//     PlcTask Inputs/GVL_iXlinker.EtherCAT_Master_BKCUCX.TcTerminals210_EK1100_1.TcTerminals210_1BK1250.A_0265_KM_2774_4_Ch_Blinds_control_CM_Inputs_230V_AC_1A.Channel_1.State <-> Channel 1/State
//     PlcTask Inputs/GVL_iXlinker.EtherCAT_Master_BKCUCX.TcTerminals210_EK1100_1.TcTerminals210_1BK1250.A_0265_KM_2774_4_Ch_Blinds_control_CM_Inputs_230V_AC_1A.Channel_1.Data_In <-> Channel 1/Data In
//     PlcTask Outputs/GVL_iXlinker.EtherCAT_Master_BKCUCX.TcTerminals210_EK1100_1.TcTerminals210_1BK1250.A_0265_KM_2774_4_Ch_Blinds_control_CM_Inputs_230V_AC_1A.Channel_1.Ctrl <-> Channel 1/Ctrl
//     PlcTask Outputs/GVL_iXlinker.EtherCAT_Master_BKCUCX.TcTerminals210_EK1100_1.TcTerminals210_1BK1250.A_0265_KM_2774_4_Ch_Blinds_control_CM_Inputs_230V_AC_1A.Channel_1.Data_Out <-> Channel 1/Data Out
//   PLC/PLC Instance <-> EtherCAT Master BKCUCX/TcTerminals210_EK1100_1/TcTerminals210_1BK1250/A_0266(Buerkert valve island 2 channels)
//     PlcTask Outputs/GVL_iXlinker.EtherCAT_Master_BKCUCX.TcTerminals210_EK1100_1.TcTerminals210_1BK1250.A_0266_Buerkert_valve_island_2_channels.Channel_1.Output <-> Channel 1/Output
//     PlcTask Outputs/GVL_iXlinker.EtherCAT_Master_BKCUCX.TcTerminals210_EK1100_1.TcTerminals210_1BK1250.A_0266_Buerkert_valve_island_2_channels.Channel_2.Output <-> Channel 2/Output
//   PLC/PLC Instance <-> EtherCAT Master BKCUCX/TcTerminals210_EK1100_1/TcTerminals210_1BK1250/A_0267(Buerkert valve island 4 channels)
//     PlcTask Outputs/GVL_iXlinker.EtherCAT_Master_BKCUCX.TcTerminals210_EK1100_1.TcTerminals210_1BK1250.A_0267_Buerkert_valve_island_4_channels.Channel_1.Output <-> Channel 1/Output
//     PlcTask Outputs/GVL_iXlinker.EtherCAT_Master_BKCUCX.TcTerminals210_EK1100_1.TcTerminals210_1BK1250.A_0267_Buerkert_valve_island_4_channels.Channel_2.Output <-> Channel 2/Output
//     PlcTask Outputs/GVL_iXlinker.EtherCAT_Master_BKCUCX.TcTerminals210_EK1100_1.TcTerminals210_1BK1250.A_0267_Buerkert_valve_island_4_channels.Channel_3.Output <-> Channel 3/Output
//     PlcTask Outputs/GVL_iXlinker.EtherCAT_Master_BKCUCX.TcTerminals210_EK1100_1.TcTerminals210_1BK1250.A_0267_Buerkert_valve_island_4_channels.Channel_4.Output <-> Channel 4/Output
//   PLC/PLC Instance <-> EtherCAT Master BKCUCX/TcTerminals210_EK1100_1/TcTerminals210_1BK1250/A_0268(Buerkert valve island 8 channels)
//     PlcTask Outputs/GVL_iXlinker.EtherCAT_Master_BKCUCX.TcTerminals210_EK1100_1.TcTerminals210_1BK1250.A_0268_Buerkert_valve_island_8_channels.Channel_1.Output <-> Channel 1/Output
//     PlcTask Outputs/GVL_iXlinker.EtherCAT_Master_BKCUCX.TcTerminals210_EK1100_1.TcTerminals210_1BK1250.A_0268_Buerkert_valve_island_8_channels.Channel_2.Output <-> Channel 2/Output
//     PlcTask Outputs/GVL_iXlinker.EtherCAT_Master_BKCUCX.TcTerminals210_EK1100_1.TcTerminals210_1BK1250.A_0268_Buerkert_valve_island_8_channels.Channel_3.Output <-> Channel 3/Output
//     PlcTask Outputs/GVL_iXlinker.EtherCAT_Master_BKCUCX.TcTerminals210_EK1100_1.TcTerminals210_1BK1250.A_0268_Buerkert_valve_island_8_channels.Channel_4.Output <-> Channel 4/Output
//     PlcTask Outputs/GVL_iXlinker.EtherCAT_Master_BKCUCX.TcTerminals210_EK1100_1.TcTerminals210_1BK1250.A_0268_Buerkert_valve_island_8_channels.Channel_5.Output <-> Channel 5/Output
//     PlcTask Outputs/GVL_iXlinker.EtherCAT_Master_BKCUCX.TcTerminals210_EK1100_1.TcTerminals210_1BK1250.A_0268_Buerkert_valve_island_8_channels.Channel_6.Output <-> Channel 6/Output
//     PlcTask Outputs/GVL_iXlinker.EtherCAT_Master_BKCUCX.TcTerminals210_EK1100_1.TcTerminals210_1BK1250.A_0268_Buerkert_valve_island_8_channels.Channel_7.Output <-> Channel 7/Output
//     PlcTask Outputs/GVL_iXlinker.EtherCAT_Master_BKCUCX.TcTerminals210_EK1100_1.TcTerminals210_1BK1250.A_0268_Buerkert_valve_island_8_channels.Channel_8.Output <-> Channel 8/Output
//   PLC/PLC Instance <-> EtherCAT Master BKCUCX/TcTerminals210_EK1100_1/TcTerminals210_1BK1250/A_0269(KL 3001, 1 Ch. ana. Input (-10V/0...10V))
//     PlcTask Inputs/GVL_iXlinker.EtherCAT_Master_BKCUCX.TcTerminals210_EK1100_1.TcTerminals210_1BK1250.A_0269_KL_3001_1_Ch_ana_Input_10V_0_10V.Channel_1.State <-> Channel 1/State
//     PlcTask Inputs/GVL_iXlinker.EtherCAT_Master_BKCUCX.TcTerminals210_EK1100_1.TcTerminals210_1BK1250.A_0269_KL_3001_1_Ch_ana_Input_10V_0_10V.Channel_1.Data_In <-> Channel 1/Data In
//     PlcTask Outputs/GVL_iXlinker.EtherCAT_Master_BKCUCX.TcTerminals210_EK1100_1.TcTerminals210_1BK1250.A_0269_KL_3001_1_Ch_ana_Input_10V_0_10V.Channel_1.Ctrl <-> Channel 1/Ctrl
//     PlcTask Outputs/GVL_iXlinker.EtherCAT_Master_BKCUCX.TcTerminals210_EK1100_1.TcTerminals210_1BK1250.A_0269_KL_3001_1_Ch_ana_Input_10V_0_10V.Channel_1.Data_Out <-> Channel 1/Data Out
//   PLC/PLC Instance <-> EtherCAT Master BKCUCX/TcTerminals210_EK1100_1/TcTerminals210_1BK1250/A_0271(KL 3002, 2 Ch. ana. Input (-10V/0...10V))
//     PlcTask Inputs/GVL_iXlinker.EtherCAT_Master_BKCUCX.TcTerminals210_EK1100_1.TcTerminals210_1BK1250.A_0271_KL_3002_2_Ch_ana_Input_10V_0_10V.Channel_1.State <-> Channel 1/State
//     PlcTask Inputs/GVL_iXlinker.EtherCAT_Master_BKCUCX.TcTerminals210_EK1100_1.TcTerminals210_1BK1250.A_0271_KL_3002_2_Ch_ana_Input_10V_0_10V.Channel_2.State <-> Channel 2/State
//     PlcTask Inputs/GVL_iXlinker.EtherCAT_Master_BKCUCX.TcTerminals210_EK1100_1.TcTerminals210_1BK1250.A_0271_KL_3002_2_Ch_ana_Input_10V_0_10V.Channel_1.Data_In <-> Channel 1/Data In
//     PlcTask Inputs/GVL_iXlinker.EtherCAT_Master_BKCUCX.TcTerminals210_EK1100_1.TcTerminals210_1BK1250.A_0271_KL_3002_2_Ch_ana_Input_10V_0_10V.Channel_2.Data_In <-> Channel 2/Data In
//     PlcTask Outputs/GVL_iXlinker.EtherCAT_Master_BKCUCX.TcTerminals210_EK1100_1.TcTerminals210_1BK1250.A_0271_KL_3002_2_Ch_ana_Input_10V_0_10V.Channel_1.Ctrl <-> Channel 1/Ctrl
//     PlcTask Outputs/GVL_iXlinker.EtherCAT_Master_BKCUCX.TcTerminals210_EK1100_1.TcTerminals210_1BK1250.A_0271_KL_3002_2_Ch_ana_Input_10V_0_10V.Channel_2.Ctrl <-> Channel 2/Ctrl
//     PlcTask Outputs/GVL_iXlinker.EtherCAT_Master_BKCUCX.TcTerminals210_EK1100_1.TcTerminals210_1BK1250.A_0271_KL_3002_2_Ch_ana_Input_10V_0_10V.Channel_1.Data_Out <-> Channel 1/Data Out
//     PlcTask Outputs/GVL_iXlinker.EtherCAT_Master_BKCUCX.TcTerminals210_EK1100_1.TcTerminals210_1BK1250.A_0271_KL_3002_2_Ch_ana_Input_10V_0_10V.Channel_2.Data_Out <-> Channel 2/Data Out
//   PLC/PLC Instance <-> EtherCAT Master BKCUCX/TcTerminals210_EK1100_1/TcTerminals210_1BK1250/A_0273(KL 3011, 1 Ch. ana. Input (0 - 20mA))
//     PlcTask Inputs/GVL_iXlinker.EtherCAT_Master_BKCUCX.TcTerminals210_EK1100_1.TcTerminals210_1BK1250.A_0273_KL_3011_1_Ch_ana_Input_0_20mA.Channel_1.State <-> Channel 1/State
//     PlcTask Inputs/GVL_iXlinker.EtherCAT_Master_BKCUCX.TcTerminals210_EK1100_1.TcTerminals210_1BK1250.A_0273_KL_3011_1_Ch_ana_Input_0_20mA.Channel_1.Data_In <-> Channel 1/Data In
//     PlcTask Outputs/GVL_iXlinker.EtherCAT_Master_BKCUCX.TcTerminals210_EK1100_1.TcTerminals210_1BK1250.A_0273_KL_3011_1_Ch_ana_Input_0_20mA.Channel_1.Ctrl <-> Channel 1/Ctrl
//     PlcTask Outputs/GVL_iXlinker.EtherCAT_Master_BKCUCX.TcTerminals210_EK1100_1.TcTerminals210_1BK1250.A_0273_KL_3011_1_Ch_ana_Input_0_20mA.Channel_1.Data_Out <-> Channel 1/Data Out
//   PLC/PLC Instance <-> EtherCAT Master BKCUCX/TcTerminals210_EK1100_1/TcTerminals210_1BK1250/A_0275(KL 3012, 2 Ch. ana. Input (0 - 20mA))
//     PlcTask Inputs/GVL_iXlinker.EtherCAT_Master_BKCUCX.TcTerminals210_EK1100_1.TcTerminals210_1BK1250.A_0275_KL_3012_2_Ch_ana_Input_0_20mA.Channel_1.State <-> Channel 1/State
//     PlcTask Inputs/GVL_iXlinker.EtherCAT_Master_BKCUCX.TcTerminals210_EK1100_1.TcTerminals210_1BK1250.A_0275_KL_3012_2_Ch_ana_Input_0_20mA.Channel_2.State <-> Channel 2/State
//     PlcTask Inputs/GVL_iXlinker.EtherCAT_Master_BKCUCX.TcTerminals210_EK1100_1.TcTerminals210_1BK1250.A_0275_KL_3012_2_Ch_ana_Input_0_20mA.Channel_1.Data_In <-> Channel 1/Data In
//     PlcTask Inputs/GVL_iXlinker.EtherCAT_Master_BKCUCX.TcTerminals210_EK1100_1.TcTerminals210_1BK1250.A_0275_KL_3012_2_Ch_ana_Input_0_20mA.Channel_2.Data_In <-> Channel 2/Data In
//     PlcTask Outputs/GVL_iXlinker.EtherCAT_Master_BKCUCX.TcTerminals210_EK1100_1.TcTerminals210_1BK1250.A_0275_KL_3012_2_Ch_ana_Input_0_20mA.Channel_1.Ctrl <-> Channel 1/Ctrl
//     PlcTask Outputs/GVL_iXlinker.EtherCAT_Master_BKCUCX.TcTerminals210_EK1100_1.TcTerminals210_1BK1250.A_0275_KL_3012_2_Ch_ana_Input_0_20mA.Channel_2.Ctrl <-> Channel 2/Ctrl
//     PlcTask Outputs/GVL_iXlinker.EtherCAT_Master_BKCUCX.TcTerminals210_EK1100_1.TcTerminals210_1BK1250.A_0275_KL_3012_2_Ch_ana_Input_0_20mA.Channel_1.Data_Out <-> Channel 1/Data Out
//     PlcTask Outputs/GVL_iXlinker.EtherCAT_Master_BKCUCX.TcTerminals210_EK1100_1.TcTerminals210_1BK1250.A_0275_KL_3012_2_Ch_ana_Input_0_20mA.Channel_2.Data_Out <-> Channel 2/Data Out
//   PLC/PLC Instance <-> EtherCAT Master BKCUCX/TcTerminals210_EK1100_1/TcTerminals210_1BK1250/A_0277(KL 3021, 1 Ch. ana. Input (4 - 20mA))
//     PlcTask Inputs/GVL_iXlinker.EtherCAT_Master_BKCUCX.TcTerminals210_EK1100_1.TcTerminals210_1BK1250.A_0277_KL_3021_1_Ch_ana_Input_4_20mA.Channel_1.State <-> Channel 1/State
//     PlcTask Inputs/GVL_iXlinker.EtherCAT_Master_BKCUCX.TcTerminals210_EK1100_1.TcTerminals210_1BK1250.A_0277_KL_3021_1_Ch_ana_Input_4_20mA.Channel_1.Data_In <-> Channel 1/Data In
//     PlcTask Outputs/GVL_iXlinker.EtherCAT_Master_BKCUCX.TcTerminals210_EK1100_1.TcTerminals210_1BK1250.A_0277_KL_3021_1_Ch_ana_Input_4_20mA.Channel_1.Ctrl <-> Channel 1/Ctrl
//     PlcTask Outputs/GVL_iXlinker.EtherCAT_Master_BKCUCX.TcTerminals210_EK1100_1.TcTerminals210_1BK1250.A_0277_KL_3021_1_Ch_ana_Input_4_20mA.Channel_1.Data_Out <-> Channel 1/Data Out
//   PLC/PLC Instance <-> EtherCAT Master BKCUCX/TcTerminals210_EK1100_1/TcTerminals210_1BK1250/A_0279(KL 3022, 2 Ch. ana. Input (4 - 20mA))
//     PlcTask Inputs/GVL_iXlinker.EtherCAT_Master_BKCUCX.TcTerminals210_EK1100_1.TcTerminals210_1BK1250.A_0279_KL_3022_2_Ch_ana_Input_4_20mA.Channel_1.State <-> Channel 1/State
//     PlcTask Inputs/GVL_iXlinker.EtherCAT_Master_BKCUCX.TcTerminals210_EK1100_1.TcTerminals210_1BK1250.A_0279_KL_3022_2_Ch_ana_Input_4_20mA.Channel_2.State <-> Channel 2/State
//     PlcTask Inputs/GVL_iXlinker.EtherCAT_Master_BKCUCX.TcTerminals210_EK1100_1.TcTerminals210_1BK1250.A_0279_KL_3022_2_Ch_ana_Input_4_20mA.Channel_1.Data_In <-> Channel 1/Data In
//     PlcTask Inputs/GVL_iXlinker.EtherCAT_Master_BKCUCX.TcTerminals210_EK1100_1.TcTerminals210_1BK1250.A_0279_KL_3022_2_Ch_ana_Input_4_20mA.Channel_2.Data_In <-> Channel 2/Data In
//     PlcTask Outputs/GVL_iXlinker.EtherCAT_Master_BKCUCX.TcTerminals210_EK1100_1.TcTerminals210_1BK1250.A_0279_KL_3022_2_Ch_ana_Input_4_20mA.Channel_1.Ctrl <-> Channel 1/Ctrl
//     PlcTask Outputs/GVL_iXlinker.EtherCAT_Master_BKCUCX.TcTerminals210_EK1100_1.TcTerminals210_1BK1250.A_0279_KL_3022_2_Ch_ana_Input_4_20mA.Channel_2.Ctrl <-> Channel 2/Ctrl
//     PlcTask Outputs/GVL_iXlinker.EtherCAT_Master_BKCUCX.TcTerminals210_EK1100_1.TcTerminals210_1BK1250.A_0279_KL_3022_2_Ch_ana_Input_4_20mA.Channel_1.Data_Out <-> Channel 1/Data Out
//     PlcTask Outputs/GVL_iXlinker.EtherCAT_Master_BKCUCX.TcTerminals210_EK1100_1.TcTerminals210_1BK1250.A_0279_KL_3022_2_Ch_ana_Input_4_20mA.Channel_2.Data_Out <-> Channel 2/Data Out
//   PLC/PLC Instance <-> EtherCAT Master BKCUCX/TcTerminals210_EK1100_1/TcTerminals210_1BK1250/A_0281(KL 3041, 1 Ch. ana. Input with Power (0 - 20mA))
//     PlcTask Inputs/GVL_iXlinker.EtherCAT_Master_BKCUCX.TcTerminals210_EK1100_1.TcTerminals210_1BK1250.A_0281_KL_3041_1_Ch_ana_Input_with_Power_0_20mA.Channel_1.State <-> Channel 1/State
//     PlcTask Inputs/GVL_iXlinker.EtherCAT_Master_BKCUCX.TcTerminals210_EK1100_1.TcTerminals210_1BK1250.A_0281_KL_3041_1_Ch_ana_Input_with_Power_0_20mA.Channel_1.Data_In <-> Channel 1/Data In
//     PlcTask Outputs/GVL_iXlinker.EtherCAT_Master_BKCUCX.TcTerminals210_EK1100_1.TcTerminals210_1BK1250.A_0281_KL_3041_1_Ch_ana_Input_with_Power_0_20mA.Channel_1.Ctrl <-> Channel 1/Ctrl
//     PlcTask Outputs/GVL_iXlinker.EtherCAT_Master_BKCUCX.TcTerminals210_EK1100_1.TcTerminals210_1BK1250.A_0281_KL_3041_1_Ch_ana_Input_with_Power_0_20mA.Channel_1.Data_Out <-> Channel 1/Data Out
//   PLC/PLC Instance <-> EtherCAT Master BKCUCX/TcTerminals210_EK1100_1/TcTerminals210_1BK1250/A_0283(KL 3042, 2 Ch. ana. Input with Power (0 - 20mA))
//     PlcTask Inputs/GVL_iXlinker.EtherCAT_Master_BKCUCX.TcTerminals210_EK1100_1.TcTerminals210_1BK1250.A_0283_KL_3042_2_Ch_ana_Input_with_Power_0_20mA.Channel_1.State <-> Channel 1/State
//     PlcTask Inputs/GVL_iXlinker.EtherCAT_Master_BKCUCX.TcTerminals210_EK1100_1.TcTerminals210_1BK1250.A_0283_KL_3042_2_Ch_ana_Input_with_Power_0_20mA.Channel_2.State <-> Channel 2/State
//     PlcTask Inputs/GVL_iXlinker.EtherCAT_Master_BKCUCX.TcTerminals210_EK1100_1.TcTerminals210_1BK1250.A_0283_KL_3042_2_Ch_ana_Input_with_Power_0_20mA.Channel_1.Data_In <-> Channel 1/Data In
//     PlcTask Inputs/GVL_iXlinker.EtherCAT_Master_BKCUCX.TcTerminals210_EK1100_1.TcTerminals210_1BK1250.A_0283_KL_3042_2_Ch_ana_Input_with_Power_0_20mA.Channel_2.Data_In <-> Channel 2/Data In
//     PlcTask Outputs/GVL_iXlinker.EtherCAT_Master_BKCUCX.TcTerminals210_EK1100_1.TcTerminals210_1BK1250.A_0283_KL_3042_2_Ch_ana_Input_with_Power_0_20mA.Channel_1.Ctrl <-> Channel 1/Ctrl
//     PlcTask Outputs/GVL_iXlinker.EtherCAT_Master_BKCUCX.TcTerminals210_EK1100_1.TcTerminals210_1BK1250.A_0283_KL_3042_2_Ch_ana_Input_with_Power_0_20mA.Channel_2.Ctrl <-> Channel 2/Ctrl
//     PlcTask Outputs/GVL_iXlinker.EtherCAT_Master_BKCUCX.TcTerminals210_EK1100_1.TcTerminals210_1BK1250.A_0283_KL_3042_2_Ch_ana_Input_with_Power_0_20mA.Channel_1.Data_Out <-> Channel 1/Data Out
//     PlcTask Outputs/GVL_iXlinker.EtherCAT_Master_BKCUCX.TcTerminals210_EK1100_1.TcTerminals210_1BK1250.A_0283_KL_3042_2_Ch_ana_Input_with_Power_0_20mA.Channel_2.Data_Out <-> Channel 2/Data Out
//   PLC/PLC Instance <-> EtherCAT Master BKCUCX/TcTerminals210_EK1100_1/TcTerminals210_1BK1250/A_0285(KL 3044, 4 Ch. ana. Input with Power (0 - 20mA))
//     PlcTask Inputs/GVL_iXlinker.EtherCAT_Master_BKCUCX.TcTerminals210_EK1100_1.TcTerminals210_1BK1250.A_0285_KL_3044_4_Ch_ana_Input_with_Power_0_20mA.Channel_1.State <-> Channel 1/State
//     PlcTask Inputs/GVL_iXlinker.EtherCAT_Master_BKCUCX.TcTerminals210_EK1100_1.TcTerminals210_1BK1250.A_0285_KL_3044_4_Ch_ana_Input_with_Power_0_20mA.Channel_2.State <-> Channel 2/State
//     PlcTask Inputs/GVL_iXlinker.EtherCAT_Master_BKCUCX.TcTerminals210_EK1100_1.TcTerminals210_1BK1250.A_0285_KL_3044_4_Ch_ana_Input_with_Power_0_20mA.Channel_3.State <-> Channel 3/State
//     PlcTask Inputs/GVL_iXlinker.EtherCAT_Master_BKCUCX.TcTerminals210_EK1100_1.TcTerminals210_1BK1250.A_0285_KL_3044_4_Ch_ana_Input_with_Power_0_20mA.Channel_4.State <-> Channel 4/State
//     PlcTask Inputs/GVL_iXlinker.EtherCAT_Master_BKCUCX.TcTerminals210_EK1100_1.TcTerminals210_1BK1250.A_0285_KL_3044_4_Ch_ana_Input_with_Power_0_20mA.Channel_1.Data_In <-> Channel 1/Data In
//     PlcTask Inputs/GVL_iXlinker.EtherCAT_Master_BKCUCX.TcTerminals210_EK1100_1.TcTerminals210_1BK1250.A_0285_KL_3044_4_Ch_ana_Input_with_Power_0_20mA.Channel_2.Data_In <-> Channel 2/Data In
//     PlcTask Inputs/GVL_iXlinker.EtherCAT_Master_BKCUCX.TcTerminals210_EK1100_1.TcTerminals210_1BK1250.A_0285_KL_3044_4_Ch_ana_Input_with_Power_0_20mA.Channel_3.Data_In <-> Channel 3/Data In
//     PlcTask Inputs/GVL_iXlinker.EtherCAT_Master_BKCUCX.TcTerminals210_EK1100_1.TcTerminals210_1BK1250.A_0285_KL_3044_4_Ch_ana_Input_with_Power_0_20mA.Channel_4.Data_In <-> Channel 4/Data In
//     PlcTask Outputs/GVL_iXlinker.EtherCAT_Master_BKCUCX.TcTerminals210_EK1100_1.TcTerminals210_1BK1250.A_0285_KL_3044_4_Ch_ana_Input_with_Power_0_20mA.Channel_1.Ctrl <-> Channel 1/Ctrl
//     PlcTask Outputs/GVL_iXlinker.EtherCAT_Master_BKCUCX.TcTerminals210_EK1100_1.TcTerminals210_1BK1250.A_0285_KL_3044_4_Ch_ana_Input_with_Power_0_20mA.Channel_2.Ctrl <-> Channel 2/Ctrl
//     PlcTask Outputs/GVL_iXlinker.EtherCAT_Master_BKCUCX.TcTerminals210_EK1100_1.TcTerminals210_1BK1250.A_0285_KL_3044_4_Ch_ana_Input_with_Power_0_20mA.Channel_3.Ctrl <-> Channel 3/Ctrl
//     PlcTask Outputs/GVL_iXlinker.EtherCAT_Master_BKCUCX.TcTerminals210_EK1100_1.TcTerminals210_1BK1250.A_0285_KL_3044_4_Ch_ana_Input_with_Power_0_20mA.Channel_4.Ctrl <-> Channel 4/Ctrl
//     PlcTask Outputs/GVL_iXlinker.EtherCAT_Master_BKCUCX.TcTerminals210_EK1100_1.TcTerminals210_1BK1250.A_0285_KL_3044_4_Ch_ana_Input_with_Power_0_20mA.Channel_1.Data_Out <-> Channel 1/Data Out
//     PlcTask Outputs/GVL_iXlinker.EtherCAT_Master_BKCUCX.TcTerminals210_EK1100_1.TcTerminals210_1BK1250.A_0285_KL_3044_4_Ch_ana_Input_with_Power_0_20mA.Channel_2.Data_Out <-> Channel 2/Data Out
//     PlcTask Outputs/GVL_iXlinker.EtherCAT_Master_BKCUCX.TcTerminals210_EK1100_1.TcTerminals210_1BK1250.A_0285_KL_3044_4_Ch_ana_Input_with_Power_0_20mA.Channel_3.Data_Out <-> Channel 3/Data Out
//     PlcTask Outputs/GVL_iXlinker.EtherCAT_Master_BKCUCX.TcTerminals210_EK1100_1.TcTerminals210_1BK1250.A_0285_KL_3044_4_Ch_ana_Input_with_Power_0_20mA.Channel_4.Data_Out <-> Channel 4/Data Out
//   PLC/PLC Instance <-> EtherCAT Master BKCUCX/TcTerminals210_EK1100_1/TcTerminals210_1BK1250/A_0287(KL 3051, 1 Ch. ana. Input with Power (4 - 20mA))
//     PlcTask Inputs/GVL_iXlinker.EtherCAT_Master_BKCUCX.TcTerminals210_EK1100_1.TcTerminals210_1BK1250.A_0287_KL_3051_1_Ch_ana_Input_with_Power_4_20mA.Channel_1.State <-> Channel 1/State
//     PlcTask Inputs/GVL_iXlinker.EtherCAT_Master_BKCUCX.TcTerminals210_EK1100_1.TcTerminals210_1BK1250.A_0287_KL_3051_1_Ch_ana_Input_with_Power_4_20mA.Channel_1.Data_In <-> Channel 1/Data In
//     PlcTask Outputs/GVL_iXlinker.EtherCAT_Master_BKCUCX.TcTerminals210_EK1100_1.TcTerminals210_1BK1250.A_0287_KL_3051_1_Ch_ana_Input_with_Power_4_20mA.Channel_1.Ctrl <-> Channel 1/Ctrl
//     PlcTask Outputs/GVL_iXlinker.EtherCAT_Master_BKCUCX.TcTerminals210_EK1100_1.TcTerminals210_1BK1250.A_0287_KL_3051_1_Ch_ana_Input_with_Power_4_20mA.Channel_1.Data_Out <-> Channel 1/Data Out
//   PLC/PLC Instance <-> EtherCAT Master BKCUCX/TcTerminals210_EK1100_1/TcTerminals210_1BK1250/A_0289(KL 3052, 2 Ch. ana. Input with Power (4 - 20mA))
//     PlcTask Inputs/GVL_iXlinker.EtherCAT_Master_BKCUCX.TcTerminals210_EK1100_1.TcTerminals210_1BK1250.A_0289_KL_3052_2_Ch_ana_Input_with_Power_4_20mA.Channel_1.State <-> Channel 1/State
//     PlcTask Inputs/GVL_iXlinker.EtherCAT_Master_BKCUCX.TcTerminals210_EK1100_1.TcTerminals210_1BK1250.A_0289_KL_3052_2_Ch_ana_Input_with_Power_4_20mA.Channel_2.State <-> Channel 2/State
//     PlcTask Inputs/GVL_iXlinker.EtherCAT_Master_BKCUCX.TcTerminals210_EK1100_1.TcTerminals210_1BK1250.A_0289_KL_3052_2_Ch_ana_Input_with_Power_4_20mA.Channel_1.Data_In <-> Channel 1/Data In
//     PlcTask Inputs/GVL_iXlinker.EtherCAT_Master_BKCUCX.TcTerminals210_EK1100_1.TcTerminals210_1BK1250.A_0289_KL_3052_2_Ch_ana_Input_with_Power_4_20mA.Channel_2.Data_In <-> Channel 2/Data In
//     PlcTask Outputs/GVL_iXlinker.EtherCAT_Master_BKCUCX.TcTerminals210_EK1100_1.TcTerminals210_1BK1250.A_0289_KL_3052_2_Ch_ana_Input_with_Power_4_20mA.Channel_1.Ctrl <-> Channel 1/Ctrl
//     PlcTask Outputs/GVL_iXlinker.EtherCAT_Master_BKCUCX.TcTerminals210_EK1100_1.TcTerminals210_1BK1250.A_0289_KL_3052_2_Ch_ana_Input_with_Power_4_20mA.Channel_2.Ctrl <-> Channel 2/Ctrl
//     PlcTask Outputs/GVL_iXlinker.EtherCAT_Master_BKCUCX.TcTerminals210_EK1100_1.TcTerminals210_1BK1250.A_0289_KL_3052_2_Ch_ana_Input_with_Power_4_20mA.Channel_1.Data_Out <-> Channel 1/Data Out
//     PlcTask Outputs/GVL_iXlinker.EtherCAT_Master_BKCUCX.TcTerminals210_EK1100_1.TcTerminals210_1BK1250.A_0289_KL_3052_2_Ch_ana_Input_with_Power_4_20mA.Channel_2.Data_Out <-> Channel 2/Data Out
//   PLC/PLC Instance <-> EtherCAT Master BKCUCX/TcTerminals210_EK1100_1/TcTerminals210_1BK1250/A_0291(KL 3054, 4 Ch. ana. Input with Power (4 - 20mA))
//     PlcTask Inputs/GVL_iXlinker.EtherCAT_Master_BKCUCX.TcTerminals210_EK1100_1.TcTerminals210_1BK1250.A_0291_KL_3054_4_Ch_ana_Input_with_Power_4_20mA.Channel_1.State <-> Channel 1/State
//     PlcTask Inputs/GVL_iXlinker.EtherCAT_Master_BKCUCX.TcTerminals210_EK1100_1.TcTerminals210_1BK1250.A_0291_KL_3054_4_Ch_ana_Input_with_Power_4_20mA.Channel_2.State <-> Channel 2/State
//     PlcTask Inputs/GVL_iXlinker.EtherCAT_Master_BKCUCX.TcTerminals210_EK1100_1.TcTerminals210_1BK1250.A_0291_KL_3054_4_Ch_ana_Input_with_Power_4_20mA.Channel_3.State <-> Channel 3/State
//     PlcTask Inputs/GVL_iXlinker.EtherCAT_Master_BKCUCX.TcTerminals210_EK1100_1.TcTerminals210_1BK1250.A_0291_KL_3054_4_Ch_ana_Input_with_Power_4_20mA.Channel_4.State <-> Channel 4/State
//     PlcTask Inputs/GVL_iXlinker.EtherCAT_Master_BKCUCX.TcTerminals210_EK1100_1.TcTerminals210_1BK1250.A_0291_KL_3054_4_Ch_ana_Input_with_Power_4_20mA.Channel_1.Data_In <-> Channel 1/Data In
//     PlcTask Inputs/GVL_iXlinker.EtherCAT_Master_BKCUCX.TcTerminals210_EK1100_1.TcTerminals210_1BK1250.A_0291_KL_3054_4_Ch_ana_Input_with_Power_4_20mA.Channel_2.Data_In <-> Channel 2/Data In
//     PlcTask Inputs/GVL_iXlinker.EtherCAT_Master_BKCUCX.TcTerminals210_EK1100_1.TcTerminals210_1BK1250.A_0291_KL_3054_4_Ch_ana_Input_with_Power_4_20mA.Channel_3.Data_In <-> Channel 3/Data In
//     PlcTask Inputs/GVL_iXlinker.EtherCAT_Master_BKCUCX.TcTerminals210_EK1100_1.TcTerminals210_1BK1250.A_0291_KL_3054_4_Ch_ana_Input_with_Power_4_20mA.Channel_4.Data_In <-> Channel 4/Data In
//     PlcTask Outputs/GVL_iXlinker.EtherCAT_Master_BKCUCX.TcTerminals210_EK1100_1.TcTerminals210_1BK1250.A_0291_KL_3054_4_Ch_ana_Input_with_Power_4_20mA.Channel_1.Ctrl <-> Channel 1/Ctrl
//     PlcTask Outputs/GVL_iXlinker.EtherCAT_Master_BKCUCX.TcTerminals210_EK1100_1.TcTerminals210_1BK1250.A_0291_KL_3054_4_Ch_ana_Input_with_Power_4_20mA.Channel_2.Ctrl <-> Channel 2/Ctrl
//     PlcTask Outputs/GVL_iXlinker.EtherCAT_Master_BKCUCX.TcTerminals210_EK1100_1.TcTerminals210_1BK1250.A_0291_KL_3054_4_Ch_ana_Input_with_Power_4_20mA.Channel_3.Ctrl <-> Channel 3/Ctrl
//     PlcTask Outputs/GVL_iXlinker.EtherCAT_Master_BKCUCX.TcTerminals210_EK1100_1.TcTerminals210_1BK1250.A_0291_KL_3054_4_Ch_ana_Input_with_Power_4_20mA.Channel_4.Ctrl <-> Channel 4/Ctrl
//     PlcTask Outputs/GVL_iXlinker.EtherCAT_Master_BKCUCX.TcTerminals210_EK1100_1.TcTerminals210_1BK1250.A_0291_KL_3054_4_Ch_ana_Input_with_Power_4_20mA.Channel_1.Data_Out <-> Channel 1/Data Out
//     PlcTask Outputs/GVL_iXlinker.EtherCAT_Master_BKCUCX.TcTerminals210_EK1100_1.TcTerminals210_1BK1250.A_0291_KL_3054_4_Ch_ana_Input_with_Power_4_20mA.Channel_2.Data_Out <-> Channel 2/Data Out
//     PlcTask Outputs/GVL_iXlinker.EtherCAT_Master_BKCUCX.TcTerminals210_EK1100_1.TcTerminals210_1BK1250.A_0291_KL_3054_4_Ch_ana_Input_with_Power_4_20mA.Channel_3.Data_Out <-> Channel 3/Data Out
//     PlcTask Outputs/GVL_iXlinker.EtherCAT_Master_BKCUCX.TcTerminals210_EK1100_1.TcTerminals210_1BK1250.A_0291_KL_3054_4_Ch_ana_Input_with_Power_4_20mA.Channel_4.Data_Out <-> Channel 4/Data Out
//   PLC/PLC Instance <-> EtherCAT Master BKCUCX/TcTerminals210_EK1100_1/TcTerminals210_1BK1250/A_0293(KL 3061, 1 Ch. ana. Input (0...10V))
//     PlcTask Inputs/GVL_iXlinker.EtherCAT_Master_BKCUCX.TcTerminals210_EK1100_1.TcTerminals210_1BK1250.A_0293_KL_3061_1_Ch_ana_Input_0_10V.Channel_1.State <-> Channel 1/State
//     PlcTask Inputs/GVL_iXlinker.EtherCAT_Master_BKCUCX.TcTerminals210_EK1100_1.TcTerminals210_1BK1250.A_0293_KL_3061_1_Ch_ana_Input_0_10V.Channel_1.Data_In <-> Channel 1/Data In
//     PlcTask Outputs/GVL_iXlinker.EtherCAT_Master_BKCUCX.TcTerminals210_EK1100_1.TcTerminals210_1BK1250.A_0293_KL_3061_1_Ch_ana_Input_0_10V.Channel_1.Ctrl <-> Channel 1/Ctrl
//     PlcTask Outputs/GVL_iXlinker.EtherCAT_Master_BKCUCX.TcTerminals210_EK1100_1.TcTerminals210_1BK1250.A_0293_KL_3061_1_Ch_ana_Input_0_10V.Channel_1.Data_Out <-> Channel 1/Data Out
//   PLC/PLC Instance <-> EtherCAT Master BKCUCX/TcTerminals210_EK1100_1/TcTerminals210_1BK1250/A_0295(KL 3062, 2 Ch. ana. Input (0...10V))
//     PlcTask Inputs/GVL_iXlinker.EtherCAT_Master_BKCUCX.TcTerminals210_EK1100_1.TcTerminals210_1BK1250.A_0295_KL_3062_2_Ch_ana_Input_0_10V.Channel_1.State <-> Channel 1/State
//     PlcTask Inputs/GVL_iXlinker.EtherCAT_Master_BKCUCX.TcTerminals210_EK1100_1.TcTerminals210_1BK1250.A_0295_KL_3062_2_Ch_ana_Input_0_10V.Channel_2.State <-> Channel 2/State
//     PlcTask Inputs/GVL_iXlinker.EtherCAT_Master_BKCUCX.TcTerminals210_EK1100_1.TcTerminals210_1BK1250.A_0295_KL_3062_2_Ch_ana_Input_0_10V.Channel_1.Data_In <-> Channel 1/Data In
//     PlcTask Inputs/GVL_iXlinker.EtherCAT_Master_BKCUCX.TcTerminals210_EK1100_1.TcTerminals210_1BK1250.A_0295_KL_3062_2_Ch_ana_Input_0_10V.Channel_2.Data_In <-> Channel 2/Data In
//     PlcTask Outputs/GVL_iXlinker.EtherCAT_Master_BKCUCX.TcTerminals210_EK1100_1.TcTerminals210_1BK1250.A_0295_KL_3062_2_Ch_ana_Input_0_10V.Channel_1.Ctrl <-> Channel 1/Ctrl
//     PlcTask Outputs/GVL_iXlinker.EtherCAT_Master_BKCUCX.TcTerminals210_EK1100_1.TcTerminals210_1BK1250.A_0295_KL_3062_2_Ch_ana_Input_0_10V.Channel_2.Ctrl <-> Channel 2/Ctrl
//     PlcTask Outputs/GVL_iXlinker.EtherCAT_Master_BKCUCX.TcTerminals210_EK1100_1.TcTerminals210_1BK1250.A_0295_KL_3062_2_Ch_ana_Input_0_10V.Channel_1.Data_Out <-> Channel 1/Data Out
//     PlcTask Outputs/GVL_iXlinker.EtherCAT_Master_BKCUCX.TcTerminals210_EK1100_1.TcTerminals210_1BK1250.A_0295_KL_3062_2_Ch_ana_Input_0_10V.Channel_2.Data_Out <-> Channel 2/Data Out
//   PLC/PLC Instance <-> EtherCAT Master BKCUCX/TcTerminals210_EK1100_1/TcTerminals210_1BK1250/A_0297(KL 3064, 4 Ch. ana. Input (0...10V))
//     PlcTask Inputs/GVL_iXlinker.EtherCAT_Master_BKCUCX.TcTerminals210_EK1100_1.TcTerminals210_1BK1250.A_0297_KL_3064_4_Ch_ana_Input_0_10V.Channel_1.State <-> Channel 1/State
//     PlcTask Inputs/GVL_iXlinker.EtherCAT_Master_BKCUCX.TcTerminals210_EK1100_1.TcTerminals210_1BK1250.A_0297_KL_3064_4_Ch_ana_Input_0_10V.Channel_2.State <-> Channel 2/State
//     PlcTask Inputs/GVL_iXlinker.EtherCAT_Master_BKCUCX.TcTerminals210_EK1100_1.TcTerminals210_1BK1250.A_0297_KL_3064_4_Ch_ana_Input_0_10V.Channel_3.State <-> Channel 3/State
//     PlcTask Inputs/GVL_iXlinker.EtherCAT_Master_BKCUCX.TcTerminals210_EK1100_1.TcTerminals210_1BK1250.A_0297_KL_3064_4_Ch_ana_Input_0_10V.Channel_4.State <-> Channel 4/State
//     PlcTask Inputs/GVL_iXlinker.EtherCAT_Master_BKCUCX.TcTerminals210_EK1100_1.TcTerminals210_1BK1250.A_0297_KL_3064_4_Ch_ana_Input_0_10V.Channel_1.Data_In <-> Channel 1/Data In
//     PlcTask Inputs/GVL_iXlinker.EtherCAT_Master_BKCUCX.TcTerminals210_EK1100_1.TcTerminals210_1BK1250.A_0297_KL_3064_4_Ch_ana_Input_0_10V.Channel_2.Data_In <-> Channel 2/Data In
//     PlcTask Inputs/GVL_iXlinker.EtherCAT_Master_BKCUCX.TcTerminals210_EK1100_1.TcTerminals210_1BK1250.A_0297_KL_3064_4_Ch_ana_Input_0_10V.Channel_3.Data_In <-> Channel 3/Data In
//     PlcTask Inputs/GVL_iXlinker.EtherCAT_Master_BKCUCX.TcTerminals210_EK1100_1.TcTerminals210_1BK1250.A_0297_KL_3064_4_Ch_ana_Input_0_10V.Channel_4.Data_In <-> Channel 4/Data In
//     PlcTask Outputs/GVL_iXlinker.EtherCAT_Master_BKCUCX.TcTerminals210_EK1100_1.TcTerminals210_1BK1250.A_0297_KL_3064_4_Ch_ana_Input_0_10V.Channel_1.Ctrl <-> Channel 1/Ctrl
//     PlcTask Outputs/GVL_iXlinker.EtherCAT_Master_BKCUCX.TcTerminals210_EK1100_1.TcTerminals210_1BK1250.A_0297_KL_3064_4_Ch_ana_Input_0_10V.Channel_2.Ctrl <-> Channel 2/Ctrl
//     PlcTask Outputs/GVL_iXlinker.EtherCAT_Master_BKCUCX.TcTerminals210_EK1100_1.TcTerminals210_1BK1250.A_0297_KL_3064_4_Ch_ana_Input_0_10V.Channel_3.Ctrl <-> Channel 3/Ctrl
//     PlcTask Outputs/GVL_iXlinker.EtherCAT_Master_BKCUCX.TcTerminals210_EK1100_1.TcTerminals210_1BK1250.A_0297_KL_3064_4_Ch_ana_Input_0_10V.Channel_4.Ctrl <-> Channel 4/Ctrl
//     PlcTask Outputs/GVL_iXlinker.EtherCAT_Master_BKCUCX.TcTerminals210_EK1100_1.TcTerminals210_1BK1250.A_0297_KL_3064_4_Ch_ana_Input_0_10V.Channel_1.Data_Out <-> Channel 1/Data Out
//     PlcTask Outputs/GVL_iXlinker.EtherCAT_Master_BKCUCX.TcTerminals210_EK1100_1.TcTerminals210_1BK1250.A_0297_KL_3064_4_Ch_ana_Input_0_10V.Channel_2.Data_Out <-> Channel 2/Data Out
//     PlcTask Outputs/GVL_iXlinker.EtherCAT_Master_BKCUCX.TcTerminals210_EK1100_1.TcTerminals210_1BK1250.A_0297_KL_3064_4_Ch_ana_Input_0_10V.Channel_3.Data_Out <-> Channel 3/Data Out
//     PlcTask Outputs/GVL_iXlinker.EtherCAT_Master_BKCUCX.TcTerminals210_EK1100_1.TcTerminals210_1BK1250.A_0297_KL_3064_4_Ch_ana_Input_0_10V.Channel_4.Data_Out <-> Channel 4/Data Out
//   PLC/PLC Instance <-> EtherCAT Master BKCUCX/TcTerminals210_EK1100_1/TcTerminals210_1BK1250/A_0299(KL 3102, 2 Ch. ana. Input 16 Bit (+/-10V))
//     PlcTask Inputs/GVL_iXlinker.EtherCAT_Master_BKCUCX.TcTerminals210_EK1100_1.TcTerminals210_1BK1250.A_0299_KL_3102_2_Ch_ana_Input_16_Bit_10V.Channel_1.State <-> Channel 1/State
//     PlcTask Inputs/GVL_iXlinker.EtherCAT_Master_BKCUCX.TcTerminals210_EK1100_1.TcTerminals210_1BK1250.A_0299_KL_3102_2_Ch_ana_Input_16_Bit_10V.Channel_2.State <-> Channel 2/State
//     PlcTask Inputs/GVL_iXlinker.EtherCAT_Master_BKCUCX.TcTerminals210_EK1100_1.TcTerminals210_1BK1250.A_0299_KL_3102_2_Ch_ana_Input_16_Bit_10V.Channel_1.Data_In <-> Channel 1/Data In
//     PlcTask Inputs/GVL_iXlinker.EtherCAT_Master_BKCUCX.TcTerminals210_EK1100_1.TcTerminals210_1BK1250.A_0299_KL_3102_2_Ch_ana_Input_16_Bit_10V.Channel_2.Data_In <-> Channel 2/Data In
//     PlcTask Outputs/GVL_iXlinker.EtherCAT_Master_BKCUCX.TcTerminals210_EK1100_1.TcTerminals210_1BK1250.A_0299_KL_3102_2_Ch_ana_Input_16_Bit_10V.Channel_1.Ctrl <-> Channel 1/Ctrl
//     PlcTask Outputs/GVL_iXlinker.EtherCAT_Master_BKCUCX.TcTerminals210_EK1100_1.TcTerminals210_1BK1250.A_0299_KL_3102_2_Ch_ana_Input_16_Bit_10V.Channel_2.Ctrl <-> Channel 2/Ctrl
//     PlcTask Outputs/GVL_iXlinker.EtherCAT_Master_BKCUCX.TcTerminals210_EK1100_1.TcTerminals210_1BK1250.A_0299_KL_3102_2_Ch_ana_Input_16_Bit_10V.Channel_1.Data_Out <-> Channel 1/Data Out
//     PlcTask Outputs/GVL_iXlinker.EtherCAT_Master_BKCUCX.TcTerminals210_EK1100_1.TcTerminals210_1BK1250.A_0299_KL_3102_2_Ch_ana_Input_16_Bit_10V.Channel_2.Data_Out <-> Channel 2/Data Out
//   PLC/PLC Instance <-> EtherCAT Master BKCUCX/TcTerminals210_EK1100_1/TcTerminals210_1BK1250/A_0301(KL 3112, 2 Ch. ana. Input 16 Bit (0 - 20mA))
//     PlcTask Inputs/GVL_iXlinker.EtherCAT_Master_BKCUCX.TcTerminals210_EK1100_1.TcTerminals210_1BK1250.A_0301_KL_3112_2_Ch_ana_Input_16_Bit_0_20mA.Channel_1.State <-> Channel 1/State
//     PlcTask Inputs/GVL_iXlinker.EtherCAT_Master_BKCUCX.TcTerminals210_EK1100_1.TcTerminals210_1BK1250.A_0301_KL_3112_2_Ch_ana_Input_16_Bit_0_20mA.Channel_2.State <-> Channel 2/State
//     PlcTask Inputs/GVL_iXlinker.EtherCAT_Master_BKCUCX.TcTerminals210_EK1100_1.TcTerminals210_1BK1250.A_0301_KL_3112_2_Ch_ana_Input_16_Bit_0_20mA.Channel_1.Data_In <-> Channel 1/Data In
//     PlcTask Inputs/GVL_iXlinker.EtherCAT_Master_BKCUCX.TcTerminals210_EK1100_1.TcTerminals210_1BK1250.A_0301_KL_3112_2_Ch_ana_Input_16_Bit_0_20mA.Channel_2.Data_In <-> Channel 2/Data In
//     PlcTask Outputs/GVL_iXlinker.EtherCAT_Master_BKCUCX.TcTerminals210_EK1100_1.TcTerminals210_1BK1250.A_0301_KL_3112_2_Ch_ana_Input_16_Bit_0_20mA.Channel_1.Ctrl <-> Channel 1/Ctrl
//     PlcTask Outputs/GVL_iXlinker.EtherCAT_Master_BKCUCX.TcTerminals210_EK1100_1.TcTerminals210_1BK1250.A_0301_KL_3112_2_Ch_ana_Input_16_Bit_0_20mA.Channel_2.Ctrl <-> Channel 2/Ctrl
//     PlcTask Outputs/GVL_iXlinker.EtherCAT_Master_BKCUCX.TcTerminals210_EK1100_1.TcTerminals210_1BK1250.A_0301_KL_3112_2_Ch_ana_Input_16_Bit_0_20mA.Channel_1.Data_Out <-> Channel 1/Data Out
//     PlcTask Outputs/GVL_iXlinker.EtherCAT_Master_BKCUCX.TcTerminals210_EK1100_1.TcTerminals210_1BK1250.A_0301_KL_3112_2_Ch_ana_Input_16_Bit_0_20mA.Channel_2.Data_Out <-> Channel 2/Data Out
//   PLC/PLC Instance <-> EtherCAT Master BKCUCX/TcTerminals210_EK1100_1/TcTerminals210_1BK1250/A_0303(KL 3122, 2 Ch. ana. Input 16 Bit (4 - 20mA))
//     PlcTask Inputs/GVL_iXlinker.EtherCAT_Master_BKCUCX.TcTerminals210_EK1100_1.TcTerminals210_1BK1250.A_0303_KL_3122_2_Ch_ana_Input_16_Bit_4_20mA.Channel_1.State <-> Channel 1/State
//     PlcTask Inputs/GVL_iXlinker.EtherCAT_Master_BKCUCX.TcTerminals210_EK1100_1.TcTerminals210_1BK1250.A_0303_KL_3122_2_Ch_ana_Input_16_Bit_4_20mA.Channel_2.State <-> Channel 2/State
//     PlcTask Inputs/GVL_iXlinker.EtherCAT_Master_BKCUCX.TcTerminals210_EK1100_1.TcTerminals210_1BK1250.A_0303_KL_3122_2_Ch_ana_Input_16_Bit_4_20mA.Channel_1.Data_In <-> Channel 1/Data In
//     PlcTask Inputs/GVL_iXlinker.EtherCAT_Master_BKCUCX.TcTerminals210_EK1100_1.TcTerminals210_1BK1250.A_0303_KL_3122_2_Ch_ana_Input_16_Bit_4_20mA.Channel_2.Data_In <-> Channel 2/Data In
//     PlcTask Outputs/GVL_iXlinker.EtherCAT_Master_BKCUCX.TcTerminals210_EK1100_1.TcTerminals210_1BK1250.A_0303_KL_3122_2_Ch_ana_Input_16_Bit_4_20mA.Channel_1.Ctrl <-> Channel 1/Ctrl
//     PlcTask Outputs/GVL_iXlinker.EtherCAT_Master_BKCUCX.TcTerminals210_EK1100_1.TcTerminals210_1BK1250.A_0303_KL_3122_2_Ch_ana_Input_16_Bit_4_20mA.Channel_2.Ctrl <-> Channel 2/Ctrl
//     PlcTask Outputs/GVL_iXlinker.EtherCAT_Master_BKCUCX.TcTerminals210_EK1100_1.TcTerminals210_1BK1250.A_0303_KL_3122_2_Ch_ana_Input_16_Bit_4_20mA.Channel_1.Data_Out <-> Channel 1/Data Out
//     PlcTask Outputs/GVL_iXlinker.EtherCAT_Master_BKCUCX.TcTerminals210_EK1100_1.TcTerminals210_1BK1250.A_0303_KL_3122_2_Ch_ana_Input_16_Bit_4_20mA.Channel_2.Data_Out <-> Channel 2/Data Out
//   PLC/PLC Instance <-> EtherCAT Master BKCUCX/TcTerminals210_EK1100_1/TcTerminals210_1BK1250/A_0305(KL 3132, 2 Ch. ana. Input 16 Bit (+/-10V))
//     PlcTask Inputs/GVL_iXlinker.EtherCAT_Master_BKCUCX.TcTerminals210_EK1100_1.TcTerminals210_1BK1250.A_0305_KL_3132_2_Ch_ana_Input_16_Bit_10V.Channel_1.State <-> Channel 1/State
//     PlcTask Inputs/GVL_iXlinker.EtherCAT_Master_BKCUCX.TcTerminals210_EK1100_1.TcTerminals210_1BK1250.A_0305_KL_3132_2_Ch_ana_Input_16_Bit_10V.Channel_2.State <-> Channel 2/State
//     PlcTask Inputs/GVL_iXlinker.EtherCAT_Master_BKCUCX.TcTerminals210_EK1100_1.TcTerminals210_1BK1250.A_0305_KL_3132_2_Ch_ana_Input_16_Bit_10V.Channel_1.Data_In <-> Channel 1/Data In
//     PlcTask Inputs/GVL_iXlinker.EtherCAT_Master_BKCUCX.TcTerminals210_EK1100_1.TcTerminals210_1BK1250.A_0305_KL_3132_2_Ch_ana_Input_16_Bit_10V.Channel_2.Data_In <-> Channel 2/Data In
//     PlcTask Outputs/GVL_iXlinker.EtherCAT_Master_BKCUCX.TcTerminals210_EK1100_1.TcTerminals210_1BK1250.A_0305_KL_3132_2_Ch_ana_Input_16_Bit_10V.Channel_1.Ctrl <-> Channel 1/Ctrl
//     PlcTask Outputs/GVL_iXlinker.EtherCAT_Master_BKCUCX.TcTerminals210_EK1100_1.TcTerminals210_1BK1250.A_0305_KL_3132_2_Ch_ana_Input_16_Bit_10V.Channel_2.Ctrl <-> Channel 2/Ctrl
//     PlcTask Outputs/GVL_iXlinker.EtherCAT_Master_BKCUCX.TcTerminals210_EK1100_1.TcTerminals210_1BK1250.A_0305_KL_3132_2_Ch_ana_Input_16_Bit_10V.Channel_1.Data_Out <-> Channel 1/Data Out
//     PlcTask Outputs/GVL_iXlinker.EtherCAT_Master_BKCUCX.TcTerminals210_EK1100_1.TcTerminals210_1BK1250.A_0305_KL_3132_2_Ch_ana_Input_16_Bit_10V.Channel_2.Data_Out <-> Channel 2/Data Out
//   PLC/PLC Instance <-> EtherCAT Master BKCUCX/TcTerminals210_EK1100_1/TcTerminals210_1BK1250/A_0307(KL 3142, 2 Ch. ana. Input with Power 16 Bit (0 - 20mA))
//     PlcTask Inputs/GVL_iXlinker.EtherCAT_Master_BKCUCX.TcTerminals210_EK1100_1.TcTerminals210_1BK1250.A_0307_KL_3142_2_Ch_ana_Input_with_Power_16_Bit_0_20mA.Channel_1.State <-> Channel 1/State
//     PlcTask Inputs/GVL_iXlinker.EtherCAT_Master_BKCUCX.TcTerminals210_EK1100_1.TcTerminals210_1BK1250.A_0307_KL_3142_2_Ch_ana_Input_with_Power_16_Bit_0_20mA.Channel_2.State <-> Channel 2/State
//     PlcTask Inputs/GVL_iXlinker.EtherCAT_Master_BKCUCX.TcTerminals210_EK1100_1.TcTerminals210_1BK1250.A_0307_KL_3142_2_Ch_ana_Input_with_Power_16_Bit_0_20mA.Channel_1.Data_In <-> Channel 1/Data In
//     PlcTask Inputs/GVL_iXlinker.EtherCAT_Master_BKCUCX.TcTerminals210_EK1100_1.TcTerminals210_1BK1250.A_0307_KL_3142_2_Ch_ana_Input_with_Power_16_Bit_0_20mA.Channel_2.Data_In <-> Channel 2/Data In
//     PlcTask Outputs/GVL_iXlinker.EtherCAT_Master_BKCUCX.TcTerminals210_EK1100_1.TcTerminals210_1BK1250.A_0307_KL_3142_2_Ch_ana_Input_with_Power_16_Bit_0_20mA.Channel_1.Ctrl <-> Channel 1/Ctrl
//     PlcTask Outputs/GVL_iXlinker.EtherCAT_Master_BKCUCX.TcTerminals210_EK1100_1.TcTerminals210_1BK1250.A_0307_KL_3142_2_Ch_ana_Input_with_Power_16_Bit_0_20mA.Channel_2.Ctrl <-> Channel 2/Ctrl
//     PlcTask Outputs/GVL_iXlinker.EtherCAT_Master_BKCUCX.TcTerminals210_EK1100_1.TcTerminals210_1BK1250.A_0307_KL_3142_2_Ch_ana_Input_with_Power_16_Bit_0_20mA.Channel_1.Data_Out <-> Channel 1/Data Out
//     PlcTask Outputs/GVL_iXlinker.EtherCAT_Master_BKCUCX.TcTerminals210_EK1100_1.TcTerminals210_1BK1250.A_0307_KL_3142_2_Ch_ana_Input_with_Power_16_Bit_0_20mA.Channel_2.Data_Out <-> Channel 2/Data Out
//   PLC/PLC Instance <-> EtherCAT Master BKCUCX/TcTerminals210_EK1100_1/TcTerminals210_1BK1250/A_0309(KL 3152, 2 Ch. ana. Input with Power 16 Bit (4 - 20mA))
//     PlcTask Inputs/GVL_iXlinker.EtherCAT_Master_BKCUCX.TcTerminals210_EK1100_1.TcTerminals210_1BK1250.A_0309_KL_3152_2_Ch_ana_Input_with_Power_16_Bit_4_20mA.Channel_1.State <-> Channel 1/State
//     PlcTask Inputs/GVL_iXlinker.EtherCAT_Master_BKCUCX.TcTerminals210_EK1100_1.TcTerminals210_1BK1250.A_0309_KL_3152_2_Ch_ana_Input_with_Power_16_Bit_4_20mA.Channel_2.State <-> Channel 2/State
//     PlcTask Inputs/GVL_iXlinker.EtherCAT_Master_BKCUCX.TcTerminals210_EK1100_1.TcTerminals210_1BK1250.A_0309_KL_3152_2_Ch_ana_Input_with_Power_16_Bit_4_20mA.Channel_1.Data_In <-> Channel 1/Data In
//     PlcTask Inputs/GVL_iXlinker.EtherCAT_Master_BKCUCX.TcTerminals210_EK1100_1.TcTerminals210_1BK1250.A_0309_KL_3152_2_Ch_ana_Input_with_Power_16_Bit_4_20mA.Channel_2.Data_In <-> Channel 2/Data In
//     PlcTask Outputs/GVL_iXlinker.EtherCAT_Master_BKCUCX.TcTerminals210_EK1100_1.TcTerminals210_1BK1250.A_0309_KL_3152_2_Ch_ana_Input_with_Power_16_Bit_4_20mA.Channel_1.Ctrl <-> Channel 1/Ctrl
//     PlcTask Outputs/GVL_iXlinker.EtherCAT_Master_BKCUCX.TcTerminals210_EK1100_1.TcTerminals210_1BK1250.A_0309_KL_3152_2_Ch_ana_Input_with_Power_16_Bit_4_20mA.Channel_2.Ctrl <-> Channel 2/Ctrl
//     PlcTask Outputs/GVL_iXlinker.EtherCAT_Master_BKCUCX.TcTerminals210_EK1100_1.TcTerminals210_1BK1250.A_0309_KL_3152_2_Ch_ana_Input_with_Power_16_Bit_4_20mA.Channel_1.Data_Out <-> Channel 1/Data Out
//     PlcTask Outputs/GVL_iXlinker.EtherCAT_Master_BKCUCX.TcTerminals210_EK1100_1.TcTerminals210_1BK1250.A_0309_KL_3152_2_Ch_ana_Input_with_Power_16_Bit_4_20mA.Channel_2.Data_Out <-> Channel 2/Data Out
//   PLC/PLC Instance <-> EtherCAT Master BKCUCX/TcTerminals210_EK1100_1/TcTerminals210_1BK1250/A_0311(KL 3158, 4 of 8 Ch. ana. Input with Power (4 - 20mA))
//     PlcTask Inputs/GVL_iXlinker.EtherCAT_Master_BKCUCX.TcTerminals210_EK1100_1.TcTerminals210_1BK1250.A_0311_KL_3158_4_of_8_Ch_ana_Input_with_Power_4_20mA.Channel_1.State <-> Channel 1/State
//     PlcTask Inputs/GVL_iXlinker.EtherCAT_Master_BKCUCX.TcTerminals210_EK1100_1.TcTerminals210_1BK1250.A_0311_KL_3158_4_of_8_Ch_ana_Input_with_Power_4_20mA.Channel_2.State <-> Channel 2/State
//     PlcTask Inputs/GVL_iXlinker.EtherCAT_Master_BKCUCX.TcTerminals210_EK1100_1.TcTerminals210_1BK1250.A_0311_KL_3158_4_of_8_Ch_ana_Input_with_Power_4_20mA.Channel_3.State <-> Channel 3/State
//     PlcTask Inputs/GVL_iXlinker.EtherCAT_Master_BKCUCX.TcTerminals210_EK1100_1.TcTerminals210_1BK1250.A_0311_KL_3158_4_of_8_Ch_ana_Input_with_Power_4_20mA.Channel_4.State <-> Channel 4/State
//     PlcTask Inputs/GVL_iXlinker.EtherCAT_Master_BKCUCX.TcTerminals210_EK1100_1.TcTerminals210_1BK1250.A_0311_KL_3158_4_of_8_Ch_ana_Input_with_Power_4_20mA.Channel_1.Data_In <-> Channel 1/Data In
//     PlcTask Inputs/GVL_iXlinker.EtherCAT_Master_BKCUCX.TcTerminals210_EK1100_1.TcTerminals210_1BK1250.A_0311_KL_3158_4_of_8_Ch_ana_Input_with_Power_4_20mA.Channel_2.Data_In <-> Channel 2/Data In
//     PlcTask Inputs/GVL_iXlinker.EtherCAT_Master_BKCUCX.TcTerminals210_EK1100_1.TcTerminals210_1BK1250.A_0311_KL_3158_4_of_8_Ch_ana_Input_with_Power_4_20mA.Channel_3.Data_In <-> Channel 3/Data In
//     PlcTask Inputs/GVL_iXlinker.EtherCAT_Master_BKCUCX.TcTerminals210_EK1100_1.TcTerminals210_1BK1250.A_0311_KL_3158_4_of_8_Ch_ana_Input_with_Power_4_20mA.Channel_4.Data_In <-> Channel 4/Data In
//     PlcTask Outputs/GVL_iXlinker.EtherCAT_Master_BKCUCX.TcTerminals210_EK1100_1.TcTerminals210_1BK1250.A_0311_KL_3158_4_of_8_Ch_ana_Input_with_Power_4_20mA.Channel_1.Ctrl <-> Channel 1/Ctrl
//     PlcTask Outputs/GVL_iXlinker.EtherCAT_Master_BKCUCX.TcTerminals210_EK1100_1.TcTerminals210_1BK1250.A_0311_KL_3158_4_of_8_Ch_ana_Input_with_Power_4_20mA.Channel_2.Ctrl <-> Channel 2/Ctrl
//     PlcTask Outputs/GVL_iXlinker.EtherCAT_Master_BKCUCX.TcTerminals210_EK1100_1.TcTerminals210_1BK1250.A_0311_KL_3158_4_of_8_Ch_ana_Input_with_Power_4_20mA.Channel_3.Ctrl <-> Channel 3/Ctrl
//     PlcTask Outputs/GVL_iXlinker.EtherCAT_Master_BKCUCX.TcTerminals210_EK1100_1.TcTerminals210_1BK1250.A_0311_KL_3158_4_of_8_Ch_ana_Input_with_Power_4_20mA.Channel_4.Ctrl <-> Channel 4/Ctrl
//     PlcTask Outputs/GVL_iXlinker.EtherCAT_Master_BKCUCX.TcTerminals210_EK1100_1.TcTerminals210_1BK1250.A_0311_KL_3158_4_of_8_Ch_ana_Input_with_Power_4_20mA.Channel_1.Data_Out <-> Channel 1/Data Out
//     PlcTask Outputs/GVL_iXlinker.EtherCAT_Master_BKCUCX.TcTerminals210_EK1100_1.TcTerminals210_1BK1250.A_0311_KL_3158_4_of_8_Ch_ana_Input_with_Power_4_20mA.Channel_2.Data_Out <-> Channel 2/Data Out
//     PlcTask Outputs/GVL_iXlinker.EtherCAT_Master_BKCUCX.TcTerminals210_EK1100_1.TcTerminals210_1BK1250.A_0311_KL_3158_4_of_8_Ch_ana_Input_with_Power_4_20mA.Channel_3.Data_Out <-> Channel 3/Data Out
//     PlcTask Outputs/GVL_iXlinker.EtherCAT_Master_BKCUCX.TcTerminals210_EK1100_1.TcTerminals210_1BK1250.A_0311_KL_3158_4_of_8_Ch_ana_Input_with_Power_4_20mA.Channel_4.Data_Out <-> Channel 4/Data Out
//   PLC/PLC Instance <-> EtherCAT Master BKCUCX/TcTerminals210_EK1100_1/TcTerminals210_1BK1250/A_0313(KL 3162, 2 Ch. ana. Input 16 Bit (0...10V))
//     PlcTask Inputs/GVL_iXlinker.EtherCAT_Master_BKCUCX.TcTerminals210_EK1100_1.TcTerminals210_1BK1250.A_0313_KL_3162_2_Ch_ana_Input_16_Bit_0_10V.Channel_1.State <-> Channel 1/State
//     PlcTask Inputs/GVL_iXlinker.EtherCAT_Master_BKCUCX.TcTerminals210_EK1100_1.TcTerminals210_1BK1250.A_0313_KL_3162_2_Ch_ana_Input_16_Bit_0_10V.Channel_2.State <-> Channel 2/State
//     PlcTask Inputs/GVL_iXlinker.EtherCAT_Master_BKCUCX.TcTerminals210_EK1100_1.TcTerminals210_1BK1250.A_0313_KL_3162_2_Ch_ana_Input_16_Bit_0_10V.Channel_1.Data_In <-> Channel 1/Data In
//     PlcTask Inputs/GVL_iXlinker.EtherCAT_Master_BKCUCX.TcTerminals210_EK1100_1.TcTerminals210_1BK1250.A_0313_KL_3162_2_Ch_ana_Input_16_Bit_0_10V.Channel_2.Data_In <-> Channel 2/Data In
//     PlcTask Outputs/GVL_iXlinker.EtherCAT_Master_BKCUCX.TcTerminals210_EK1100_1.TcTerminals210_1BK1250.A_0313_KL_3162_2_Ch_ana_Input_16_Bit_0_10V.Channel_1.Ctrl <-> Channel 1/Ctrl
//     PlcTask Outputs/GVL_iXlinker.EtherCAT_Master_BKCUCX.TcTerminals210_EK1100_1.TcTerminals210_1BK1250.A_0313_KL_3162_2_Ch_ana_Input_16_Bit_0_10V.Channel_2.Ctrl <-> Channel 2/Ctrl
//     PlcTask Outputs/GVL_iXlinker.EtherCAT_Master_BKCUCX.TcTerminals210_EK1100_1.TcTerminals210_1BK1250.A_0313_KL_3162_2_Ch_ana_Input_16_Bit_0_10V.Channel_1.Data_Out <-> Channel 1/Data Out
//     PlcTask Outputs/GVL_iXlinker.EtherCAT_Master_BKCUCX.TcTerminals210_EK1100_1.TcTerminals210_1BK1250.A_0313_KL_3162_2_Ch_ana_Input_16_Bit_0_10V.Channel_2.Data_Out <-> Channel 2/Data Out
//   PLC/PLC Instance <-> EtherCAT Master BKCUCX/TcTerminals210_EK1100_1/TcTerminals210_1BK1250/A_0315(KL 3172, 2 Ch. ana. Input 16 Bit (0-2V))
//     PlcTask Inputs/GVL_iXlinker.EtherCAT_Master_BKCUCX.TcTerminals210_EK1100_1.TcTerminals210_1BK1250.A_0315_KL_3172_2_Ch_ana_Input_16_Bit_0_2V.Channel_1.State <-> Channel 1/State
//     PlcTask Inputs/GVL_iXlinker.EtherCAT_Master_BKCUCX.TcTerminals210_EK1100_1.TcTerminals210_1BK1250.A_0315_KL_3172_2_Ch_ana_Input_16_Bit_0_2V.Channel_2.State <-> Channel 2/State
//     PlcTask Inputs/GVL_iXlinker.EtherCAT_Master_BKCUCX.TcTerminals210_EK1100_1.TcTerminals210_1BK1250.A_0315_KL_3172_2_Ch_ana_Input_16_Bit_0_2V.Channel_1.Data_In <-> Channel 1/Data In
//     PlcTask Inputs/GVL_iXlinker.EtherCAT_Master_BKCUCX.TcTerminals210_EK1100_1.TcTerminals210_1BK1250.A_0315_KL_3172_2_Ch_ana_Input_16_Bit_0_2V.Channel_2.Data_In <-> Channel 2/Data In
//     PlcTask Outputs/GVL_iXlinker.EtherCAT_Master_BKCUCX.TcTerminals210_EK1100_1.TcTerminals210_1BK1250.A_0315_KL_3172_2_Ch_ana_Input_16_Bit_0_2V.Channel_1.Ctrl <-> Channel 1/Ctrl
//     PlcTask Outputs/GVL_iXlinker.EtherCAT_Master_BKCUCX.TcTerminals210_EK1100_1.TcTerminals210_1BK1250.A_0315_KL_3172_2_Ch_ana_Input_16_Bit_0_2V.Channel_2.Ctrl <-> Channel 2/Ctrl
//     PlcTask Outputs/GVL_iXlinker.EtherCAT_Master_BKCUCX.TcTerminals210_EK1100_1.TcTerminals210_1BK1250.A_0315_KL_3172_2_Ch_ana_Input_16_Bit_0_2V.Channel_1.Data_Out <-> Channel 1/Data Out
//     PlcTask Outputs/GVL_iXlinker.EtherCAT_Master_BKCUCX.TcTerminals210_EK1100_1.TcTerminals210_1BK1250.A_0315_KL_3172_2_Ch_ana_Input_16_Bit_0_2V.Channel_2.Data_Out <-> Channel 2/Data Out
//   PLC/PLC Instance <-> EtherCAT Master BKCUCX/TcTerminals210_EK1100_1/TcTerminals210_1BK1250/A_0317(KL 3172-0500, 2 Ch. ana. Input 16 Bit (0-0.5V))
//     PlcTask Inputs/GVL_iXlinker.EtherCAT_Master_BKCUCX.TcTerminals210_EK1100_1.TcTerminals210_1BK1250.A_0317_KL_3172_0500_2_Ch_ana_Input_16_Bit_0_0_5V.Channel_1.State <-> Channel 1/State
//     PlcTask Inputs/GVL_iXlinker.EtherCAT_Master_BKCUCX.TcTerminals210_EK1100_1.TcTerminals210_1BK1250.A_0317_KL_3172_0500_2_Ch_ana_Input_16_Bit_0_0_5V.Channel_2.State <-> Channel 2/State
//     PlcTask Inputs/GVL_iXlinker.EtherCAT_Master_BKCUCX.TcTerminals210_EK1100_1.TcTerminals210_1BK1250.A_0317_KL_3172_0500_2_Ch_ana_Input_16_Bit_0_0_5V.Channel_1.Data_In <-> Channel 1/Data In
//     PlcTask Inputs/GVL_iXlinker.EtherCAT_Master_BKCUCX.TcTerminals210_EK1100_1.TcTerminals210_1BK1250.A_0317_KL_3172_0500_2_Ch_ana_Input_16_Bit_0_0_5V.Channel_2.Data_In <-> Channel 2/Data In
//     PlcTask Outputs/GVL_iXlinker.EtherCAT_Master_BKCUCX.TcTerminals210_EK1100_1.TcTerminals210_1BK1250.A_0317_KL_3172_0500_2_Ch_ana_Input_16_Bit_0_0_5V.Channel_1.Ctrl <-> Channel 1/Ctrl
//     PlcTask Outputs/GVL_iXlinker.EtherCAT_Master_BKCUCX.TcTerminals210_EK1100_1.TcTerminals210_1BK1250.A_0317_KL_3172_0500_2_Ch_ana_Input_16_Bit_0_0_5V.Channel_2.Ctrl <-> Channel 2/Ctrl
//     PlcTask Outputs/GVL_iXlinker.EtherCAT_Master_BKCUCX.TcTerminals210_EK1100_1.TcTerminals210_1BK1250.A_0317_KL_3172_0500_2_Ch_ana_Input_16_Bit_0_0_5V.Channel_1.Data_Out <-> Channel 1/Data Out
//     PlcTask Outputs/GVL_iXlinker.EtherCAT_Master_BKCUCX.TcTerminals210_EK1100_1.TcTerminals210_1BK1250.A_0317_KL_3172_0500_2_Ch_ana_Input_16_Bit_0_0_5V.Channel_2.Data_Out <-> Channel 2/Data Out
//   PLC/PLC Instance <-> EtherCAT Master BKCUCX/TcTerminals210_EK1100_1/TcTerminals210_1BK1250/A_0319(KL 3172-1000, 2 Ch. ana. Input 16 Bit (0-1V))
//     PlcTask Inputs/GVL_iXlinker.EtherCAT_Master_BKCUCX.TcTerminals210_EK1100_1.TcTerminals210_1BK1250.A_0319_KL_3172_1000_2_Ch_ana_Input_16_Bit_0_1V.Channel_1.State <-> Channel 1/State
//     PlcTask Inputs/GVL_iXlinker.EtherCAT_Master_BKCUCX.TcTerminals210_EK1100_1.TcTerminals210_1BK1250.A_0319_KL_3172_1000_2_Ch_ana_Input_16_Bit_0_1V.Channel_2.State <-> Channel 2/State
//     PlcTask Inputs/GVL_iXlinker.EtherCAT_Master_BKCUCX.TcTerminals210_EK1100_1.TcTerminals210_1BK1250.A_0319_KL_3172_1000_2_Ch_ana_Input_16_Bit_0_1V.Channel_1.Data_In <-> Channel 1/Data In
//     PlcTask Inputs/GVL_iXlinker.EtherCAT_Master_BKCUCX.TcTerminals210_EK1100_1.TcTerminals210_1BK1250.A_0319_KL_3172_1000_2_Ch_ana_Input_16_Bit_0_1V.Channel_2.Data_In <-> Channel 2/Data In
//     PlcTask Outputs/GVL_iXlinker.EtherCAT_Master_BKCUCX.TcTerminals210_EK1100_1.TcTerminals210_1BK1250.A_0319_KL_3172_1000_2_Ch_ana_Input_16_Bit_0_1V.Channel_1.Ctrl <-> Channel 1/Ctrl
//     PlcTask Outputs/GVL_iXlinker.EtherCAT_Master_BKCUCX.TcTerminals210_EK1100_1.TcTerminals210_1BK1250.A_0319_KL_3172_1000_2_Ch_ana_Input_16_Bit_0_1V.Channel_2.Ctrl <-> Channel 2/Ctrl
//     PlcTask Outputs/GVL_iXlinker.EtherCAT_Master_BKCUCX.TcTerminals210_EK1100_1.TcTerminals210_1BK1250.A_0319_KL_3172_1000_2_Ch_ana_Input_16_Bit_0_1V.Channel_1.Data_Out <-> Channel 1/Data Out
//     PlcTask Outputs/GVL_iXlinker.EtherCAT_Master_BKCUCX.TcTerminals210_EK1100_1.TcTerminals210_1BK1250.A_0319_KL_3172_1000_2_Ch_ana_Input_16_Bit_0_1V.Channel_2.Data_Out <-> Channel 2/Data Out
//   PLC/PLC Instance <-> EtherCAT Master BKCUCX/TcTerminals210_EK1100_1/TcTerminals210_1BK1250/A_0321(KL 3182, 2 Ch. ana. Input 16 Bit (+/-2V))
//     PlcTask Inputs/GVL_iXlinker.EtherCAT_Master_BKCUCX.TcTerminals210_EK1100_1.TcTerminals210_1BK1250.A_0321_KL_3182_2_Ch_ana_Input_16_Bit_2V.Channel_1.State <-> Channel 1/State
//     PlcTask Inputs/GVL_iXlinker.EtherCAT_Master_BKCUCX.TcTerminals210_EK1100_1.TcTerminals210_1BK1250.A_0321_KL_3182_2_Ch_ana_Input_16_Bit_2V.Channel_2.State <-> Channel 2/State
//     PlcTask Inputs/GVL_iXlinker.EtherCAT_Master_BKCUCX.TcTerminals210_EK1100_1.TcTerminals210_1BK1250.A_0321_KL_3182_2_Ch_ana_Input_16_Bit_2V.Channel_1.Data_In <-> Channel 1/Data In
//     PlcTask Inputs/GVL_iXlinker.EtherCAT_Master_BKCUCX.TcTerminals210_EK1100_1.TcTerminals210_1BK1250.A_0321_KL_3182_2_Ch_ana_Input_16_Bit_2V.Channel_2.Data_In <-> Channel 2/Data In
//     PlcTask Outputs/GVL_iXlinker.EtherCAT_Master_BKCUCX.TcTerminals210_EK1100_1.TcTerminals210_1BK1250.A_0321_KL_3182_2_Ch_ana_Input_16_Bit_2V.Channel_1.Ctrl <-> Channel 1/Ctrl
//     PlcTask Outputs/GVL_iXlinker.EtherCAT_Master_BKCUCX.TcTerminals210_EK1100_1.TcTerminals210_1BK1250.A_0321_KL_3182_2_Ch_ana_Input_16_Bit_2V.Channel_2.Ctrl <-> Channel 2/Ctrl
//     PlcTask Outputs/GVL_iXlinker.EtherCAT_Master_BKCUCX.TcTerminals210_EK1100_1.TcTerminals210_1BK1250.A_0321_KL_3182_2_Ch_ana_Input_16_Bit_2V.Channel_1.Data_Out <-> Channel 1/Data Out
//     PlcTask Outputs/GVL_iXlinker.EtherCAT_Master_BKCUCX.TcTerminals210_EK1100_1.TcTerminals210_1BK1250.A_0321_KL_3182_2_Ch_ana_Input_16_Bit_2V.Channel_2.Data_Out <-> Channel 2/Data Out
//   PLC/PLC Instance <-> EtherCAT Master BKCUCX/TcTerminals210_EK1100_1/TcTerminals210_1BK1250/A_0323(KL 3201, 1 Ch. ana. Input PT100 (RTD))
//     PlcTask Inputs/GVL_iXlinker.EtherCAT_Master_BKCUCX.TcTerminals210_EK1100_1.TcTerminals210_1BK1250.A_0323_KL_3201_1_Ch_ana_Input_PT100_RTD.Channel_1.State <-> Channel 1/State
//     PlcTask Inputs/GVL_iXlinker.EtherCAT_Master_BKCUCX.TcTerminals210_EK1100_1.TcTerminals210_1BK1250.A_0323_KL_3201_1_Ch_ana_Input_PT100_RTD.Channel_1.Data_In <-> Channel 1/Data In
//     PlcTask Outputs/GVL_iXlinker.EtherCAT_Master_BKCUCX.TcTerminals210_EK1100_1.TcTerminals210_1BK1250.A_0323_KL_3201_1_Ch_ana_Input_PT100_RTD.Channel_1.Ctrl <-> Channel 1/Ctrl
//     PlcTask Outputs/GVL_iXlinker.EtherCAT_Master_BKCUCX.TcTerminals210_EK1100_1.TcTerminals210_1BK1250.A_0323_KL_3201_1_Ch_ana_Input_PT100_RTD.Channel_1.Data_Out <-> Channel 1/Data Out
//   PLC/PLC Instance <-> EtherCAT Master BKCUCX/TcTerminals210_EK1100_1/TcTerminals210_1BK1250/A_0325(KL 3202, 2 Ch. ana. Input PT100 (RTD))
//     PlcTask Inputs/GVL_iXlinker.EtherCAT_Master_BKCUCX.TcTerminals210_EK1100_1.TcTerminals210_1BK1250.A_0325_KL_3202_2_Ch_ana_Input_PT100_RTD.Channel_1.State <-> Channel 1/State
//     PlcTask Inputs/GVL_iXlinker.EtherCAT_Master_BKCUCX.TcTerminals210_EK1100_1.TcTerminals210_1BK1250.A_0325_KL_3202_2_Ch_ana_Input_PT100_RTD.Channel_2.State <-> Channel 2/State
//     PlcTask Inputs/GVL_iXlinker.EtherCAT_Master_BKCUCX.TcTerminals210_EK1100_1.TcTerminals210_1BK1250.A_0325_KL_3202_2_Ch_ana_Input_PT100_RTD.Channel_1.Data_In <-> Channel 1/Data In
//     PlcTask Inputs/GVL_iXlinker.EtherCAT_Master_BKCUCX.TcTerminals210_EK1100_1.TcTerminals210_1BK1250.A_0325_KL_3202_2_Ch_ana_Input_PT100_RTD.Channel_2.Data_In <-> Channel 2/Data In
//     PlcTask Outputs/GVL_iXlinker.EtherCAT_Master_BKCUCX.TcTerminals210_EK1100_1.TcTerminals210_1BK1250.A_0325_KL_3202_2_Ch_ana_Input_PT100_RTD.Channel_1.Ctrl <-> Channel 1/Ctrl
//     PlcTask Outputs/GVL_iXlinker.EtherCAT_Master_BKCUCX.TcTerminals210_EK1100_1.TcTerminals210_1BK1250.A_0325_KL_3202_2_Ch_ana_Input_PT100_RTD.Channel_2.Ctrl <-> Channel 2/Ctrl
//     PlcTask Outputs/GVL_iXlinker.EtherCAT_Master_BKCUCX.TcTerminals210_EK1100_1.TcTerminals210_1BK1250.A_0325_KL_3202_2_Ch_ana_Input_PT100_RTD.Channel_1.Data_Out <-> Channel 1/Data Out
//     PlcTask Outputs/GVL_iXlinker.EtherCAT_Master_BKCUCX.TcTerminals210_EK1100_1.TcTerminals210_1BK1250.A_0325_KL_3202_2_Ch_ana_Input_PT100_RTD.Channel_2.Data_Out <-> Channel 2/Data Out
//   PLC/PLC Instance <-> EtherCAT Master BKCUCX/TcTerminals210_EK1100_1/TcTerminals210_1BK1250/A_0327(KL 3204, 4 Ch. ana. Input PT100 (RTD))
//     PlcTask Inputs/GVL_iXlinker.EtherCAT_Master_BKCUCX.TcTerminals210_EK1100_1.TcTerminals210_1BK1250.A_0327_KL_3204_4_Ch_ana_Input_PT100_RTD.Channel_1.State <-> Channel 1/State
//     PlcTask Inputs/GVL_iXlinker.EtherCAT_Master_BKCUCX.TcTerminals210_EK1100_1.TcTerminals210_1BK1250.A_0327_KL_3204_4_Ch_ana_Input_PT100_RTD.Channel_2.State <-> Channel 2/State
//     PlcTask Inputs/GVL_iXlinker.EtherCAT_Master_BKCUCX.TcTerminals210_EK1100_1.TcTerminals210_1BK1250.A_0327_KL_3204_4_Ch_ana_Input_PT100_RTD.Channel_3.State <-> Channel 3/State
//     PlcTask Inputs/GVL_iXlinker.EtherCAT_Master_BKCUCX.TcTerminals210_EK1100_1.TcTerminals210_1BK1250.A_0327_KL_3204_4_Ch_ana_Input_PT100_RTD.Channel_4.State <-> Channel 4/State
//     PlcTask Inputs/GVL_iXlinker.EtherCAT_Master_BKCUCX.TcTerminals210_EK1100_1.TcTerminals210_1BK1250.A_0327_KL_3204_4_Ch_ana_Input_PT100_RTD.Channel_1.Data_In <-> Channel 1/Data In
//     PlcTask Inputs/GVL_iXlinker.EtherCAT_Master_BKCUCX.TcTerminals210_EK1100_1.TcTerminals210_1BK1250.A_0327_KL_3204_4_Ch_ana_Input_PT100_RTD.Channel_2.Data_In <-> Channel 2/Data In
//     PlcTask Inputs/GVL_iXlinker.EtherCAT_Master_BKCUCX.TcTerminals210_EK1100_1.TcTerminals210_1BK1250.A_0327_KL_3204_4_Ch_ana_Input_PT100_RTD.Channel_3.Data_In <-> Channel 3/Data In
//     PlcTask Inputs/GVL_iXlinker.EtherCAT_Master_BKCUCX.TcTerminals210_EK1100_1.TcTerminals210_1BK1250.A_0327_KL_3204_4_Ch_ana_Input_PT100_RTD.Channel_4.Data_In <-> Channel 4/Data In
//     PlcTask Outputs/GVL_iXlinker.EtherCAT_Master_BKCUCX.TcTerminals210_EK1100_1.TcTerminals210_1BK1250.A_0327_KL_3204_4_Ch_ana_Input_PT100_RTD.Channel_1.Ctrl <-> Channel 1/Ctrl
//     PlcTask Outputs/GVL_iXlinker.EtherCAT_Master_BKCUCX.TcTerminals210_EK1100_1.TcTerminals210_1BK1250.A_0327_KL_3204_4_Ch_ana_Input_PT100_RTD.Channel_2.Ctrl <-> Channel 2/Ctrl
//     PlcTask Outputs/GVL_iXlinker.EtherCAT_Master_BKCUCX.TcTerminals210_EK1100_1.TcTerminals210_1BK1250.A_0327_KL_3204_4_Ch_ana_Input_PT100_RTD.Channel_3.Ctrl <-> Channel 3/Ctrl
//     PlcTask Outputs/GVL_iXlinker.EtherCAT_Master_BKCUCX.TcTerminals210_EK1100_1.TcTerminals210_1BK1250.A_0327_KL_3204_4_Ch_ana_Input_PT100_RTD.Channel_4.Ctrl <-> Channel 4/Ctrl
//     PlcTask Outputs/GVL_iXlinker.EtherCAT_Master_BKCUCX.TcTerminals210_EK1100_1.TcTerminals210_1BK1250.A_0327_KL_3204_4_Ch_ana_Input_PT100_RTD.Channel_1.Data_Out <-> Channel 1/Data Out
//     PlcTask Outputs/GVL_iXlinker.EtherCAT_Master_BKCUCX.TcTerminals210_EK1100_1.TcTerminals210_1BK1250.A_0327_KL_3204_4_Ch_ana_Input_PT100_RTD.Channel_2.Data_Out <-> Channel 2/Data Out
//     PlcTask Outputs/GVL_iXlinker.EtherCAT_Master_BKCUCX.TcTerminals210_EK1100_1.TcTerminals210_1BK1250.A_0327_KL_3204_4_Ch_ana_Input_PT100_RTD.Channel_3.Data_Out <-> Channel 3/Data Out
//     PlcTask Outputs/GVL_iXlinker.EtherCAT_Master_BKCUCX.TcTerminals210_EK1100_1.TcTerminals210_1BK1250.A_0327_KL_3204_4_Ch_ana_Input_PT100_RTD.Channel_4.Data_Out <-> Channel 4/Data Out
//   PLC/PLC Instance <-> EtherCAT Master BKCUCX/TcTerminals210_EK1100_1/TcTerminals210_1BK1250/A_0329(KL 3208-0010, 4 of 8 Ch. ana. Input PT1000, Ni1000 (RTD))
//     PlcTask Inputs/GVL_iXlinker.EtherCAT_Master_BKCUCX.TcTerminals210_EK1100_1.TcTerminals210_1BK1250.A_0329_KL_3208_0010_4_of_8_Ch_ana_Input_PT1000_Ni1000_RTD.Channel_1.State <-> Channel 1/State
//     PlcTask Inputs/GVL_iXlinker.EtherCAT_Master_BKCUCX.TcTerminals210_EK1100_1.TcTerminals210_1BK1250.A_0329_KL_3208_0010_4_of_8_Ch_ana_Input_PT1000_Ni1000_RTD.Channel_2.State <-> Channel 2/State
//     PlcTask Inputs/GVL_iXlinker.EtherCAT_Master_BKCUCX.TcTerminals210_EK1100_1.TcTerminals210_1BK1250.A_0329_KL_3208_0010_4_of_8_Ch_ana_Input_PT1000_Ni1000_RTD.Channel_3.State <-> Channel 3/State
//     PlcTask Inputs/GVL_iXlinker.EtherCAT_Master_BKCUCX.TcTerminals210_EK1100_1.TcTerminals210_1BK1250.A_0329_KL_3208_0010_4_of_8_Ch_ana_Input_PT1000_Ni1000_RTD.Channel_4.State <-> Channel 4/State
//     PlcTask Inputs/GVL_iXlinker.EtherCAT_Master_BKCUCX.TcTerminals210_EK1100_1.TcTerminals210_1BK1250.A_0329_KL_3208_0010_4_of_8_Ch_ana_Input_PT1000_Ni1000_RTD.Channel_1.Data_In <-> Channel 1/Data In
//     PlcTask Inputs/GVL_iXlinker.EtherCAT_Master_BKCUCX.TcTerminals210_EK1100_1.TcTerminals210_1BK1250.A_0329_KL_3208_0010_4_of_8_Ch_ana_Input_PT1000_Ni1000_RTD.Channel_2.Data_In <-> Channel 2/Data In
//     PlcTask Inputs/GVL_iXlinker.EtherCAT_Master_BKCUCX.TcTerminals210_EK1100_1.TcTerminals210_1BK1250.A_0329_KL_3208_0010_4_of_8_Ch_ana_Input_PT1000_Ni1000_RTD.Channel_3.Data_In <-> Channel 3/Data In
//     PlcTask Inputs/GVL_iXlinker.EtherCAT_Master_BKCUCX.TcTerminals210_EK1100_1.TcTerminals210_1BK1250.A_0329_KL_3208_0010_4_of_8_Ch_ana_Input_PT1000_Ni1000_RTD.Channel_4.Data_In <-> Channel 4/Data In
//     PlcTask Outputs/GVL_iXlinker.EtherCAT_Master_BKCUCX.TcTerminals210_EK1100_1.TcTerminals210_1BK1250.A_0329_KL_3208_0010_4_of_8_Ch_ana_Input_PT1000_Ni1000_RTD.Channel_1.Ctrl <-> Channel 1/Ctrl
//     PlcTask Outputs/GVL_iXlinker.EtherCAT_Master_BKCUCX.TcTerminals210_EK1100_1.TcTerminals210_1BK1250.A_0329_KL_3208_0010_4_of_8_Ch_ana_Input_PT1000_Ni1000_RTD.Channel_2.Ctrl <-> Channel 2/Ctrl
//     PlcTask Outputs/GVL_iXlinker.EtherCAT_Master_BKCUCX.TcTerminals210_EK1100_1.TcTerminals210_1BK1250.A_0329_KL_3208_0010_4_of_8_Ch_ana_Input_PT1000_Ni1000_RTD.Channel_3.Ctrl <-> Channel 3/Ctrl
//     PlcTask Outputs/GVL_iXlinker.EtherCAT_Master_BKCUCX.TcTerminals210_EK1100_1.TcTerminals210_1BK1250.A_0329_KL_3208_0010_4_of_8_Ch_ana_Input_PT1000_Ni1000_RTD.Channel_4.Ctrl <-> Channel 4/Ctrl
//     PlcTask Outputs/GVL_iXlinker.EtherCAT_Master_BKCUCX.TcTerminals210_EK1100_1.TcTerminals210_1BK1250.A_0329_KL_3208_0010_4_of_8_Ch_ana_Input_PT1000_Ni1000_RTD.Channel_1.Data_Out <-> Channel 1/Data Out
//     PlcTask Outputs/GVL_iXlinker.EtherCAT_Master_BKCUCX.TcTerminals210_EK1100_1.TcTerminals210_1BK1250.A_0329_KL_3208_0010_4_of_8_Ch_ana_Input_PT1000_Ni1000_RTD.Channel_2.Data_Out <-> Channel 2/Data Out
//     PlcTask Outputs/GVL_iXlinker.EtherCAT_Master_BKCUCX.TcTerminals210_EK1100_1.TcTerminals210_1BK1250.A_0329_KL_3208_0010_4_of_8_Ch_ana_Input_PT1000_Ni1000_RTD.Channel_3.Data_Out <-> Channel 3/Data Out
//     PlcTask Outputs/GVL_iXlinker.EtherCAT_Master_BKCUCX.TcTerminals210_EK1100_1.TcTerminals210_1BK1250.A_0329_KL_3208_0010_4_of_8_Ch_ana_Input_PT1000_Ni1000_RTD.Channel_4.Data_Out <-> Channel 4/Data Out
//   PLC/PLC Instance <-> EtherCAT Master BKCUCX/TcTerminals210_EK1100_1/TcTerminals210_1BK1250/A_0331(KL 3214, 4 Ch. ana. Input PT100 (RTD, 3 wire))
//     PlcTask Inputs/GVL_iXlinker.EtherCAT_Master_BKCUCX.TcTerminals210_EK1100_1.TcTerminals210_1BK1250.A_0331_KL_3214_4_Ch_ana_Input_PT100_RTD_3_wire.Channel_1.State <-> Channel 1/State
//     PlcTask Inputs/GVL_iXlinker.EtherCAT_Master_BKCUCX.TcTerminals210_EK1100_1.TcTerminals210_1BK1250.A_0331_KL_3214_4_Ch_ana_Input_PT100_RTD_3_wire.Channel_2.State <-> Channel 2/State
//     PlcTask Inputs/GVL_iXlinker.EtherCAT_Master_BKCUCX.TcTerminals210_EK1100_1.TcTerminals210_1BK1250.A_0331_KL_3214_4_Ch_ana_Input_PT100_RTD_3_wire.Channel_3.State <-> Channel 3/State
//     PlcTask Inputs/GVL_iXlinker.EtherCAT_Master_BKCUCX.TcTerminals210_EK1100_1.TcTerminals210_1BK1250.A_0331_KL_3214_4_Ch_ana_Input_PT100_RTD_3_wire.Channel_4.State <-> Channel 4/State
//     PlcTask Inputs/GVL_iXlinker.EtherCAT_Master_BKCUCX.TcTerminals210_EK1100_1.TcTerminals210_1BK1250.A_0331_KL_3214_4_Ch_ana_Input_PT100_RTD_3_wire.Channel_1.Data_In <-> Channel 1/Data In
//     PlcTask Inputs/GVL_iXlinker.EtherCAT_Master_BKCUCX.TcTerminals210_EK1100_1.TcTerminals210_1BK1250.A_0331_KL_3214_4_Ch_ana_Input_PT100_RTD_3_wire.Channel_2.Data_In <-> Channel 2/Data In
//     PlcTask Inputs/GVL_iXlinker.EtherCAT_Master_BKCUCX.TcTerminals210_EK1100_1.TcTerminals210_1BK1250.A_0331_KL_3214_4_Ch_ana_Input_PT100_RTD_3_wire.Channel_3.Data_In <-> Channel 3/Data In
//     PlcTask Inputs/GVL_iXlinker.EtherCAT_Master_BKCUCX.TcTerminals210_EK1100_1.TcTerminals210_1BK1250.A_0331_KL_3214_4_Ch_ana_Input_PT100_RTD_3_wire.Channel_4.Data_In <-> Channel 4/Data In
//     PlcTask Outputs/GVL_iXlinker.EtherCAT_Master_BKCUCX.TcTerminals210_EK1100_1.TcTerminals210_1BK1250.A_0331_KL_3214_4_Ch_ana_Input_PT100_RTD_3_wire.Channel_1.Ctrl <-> Channel 1/Ctrl
//     PlcTask Outputs/GVL_iXlinker.EtherCAT_Master_BKCUCX.TcTerminals210_EK1100_1.TcTerminals210_1BK1250.A_0331_KL_3214_4_Ch_ana_Input_PT100_RTD_3_wire.Channel_2.Ctrl <-> Channel 2/Ctrl
//     PlcTask Outputs/GVL_iXlinker.EtherCAT_Master_BKCUCX.TcTerminals210_EK1100_1.TcTerminals210_1BK1250.A_0331_KL_3214_4_Ch_ana_Input_PT100_RTD_3_wire.Channel_3.Ctrl <-> Channel 3/Ctrl
//     PlcTask Outputs/GVL_iXlinker.EtherCAT_Master_BKCUCX.TcTerminals210_EK1100_1.TcTerminals210_1BK1250.A_0331_KL_3214_4_Ch_ana_Input_PT100_RTD_3_wire.Channel_4.Ctrl <-> Channel 4/Ctrl
//     PlcTask Outputs/GVL_iXlinker.EtherCAT_Master_BKCUCX.TcTerminals210_EK1100_1.TcTerminals210_1BK1250.A_0331_KL_3214_4_Ch_ana_Input_PT100_RTD_3_wire.Channel_1.Data_Out <-> Channel 1/Data Out
//     PlcTask Outputs/GVL_iXlinker.EtherCAT_Master_BKCUCX.TcTerminals210_EK1100_1.TcTerminals210_1BK1250.A_0331_KL_3214_4_Ch_ana_Input_PT100_RTD_3_wire.Channel_2.Data_Out <-> Channel 2/Data Out
//     PlcTask Outputs/GVL_iXlinker.EtherCAT_Master_BKCUCX.TcTerminals210_EK1100_1.TcTerminals210_1BK1250.A_0331_KL_3214_4_Ch_ana_Input_PT100_RTD_3_wire.Channel_3.Data_Out <-> Channel 3/Data Out
//     PlcTask Outputs/GVL_iXlinker.EtherCAT_Master_BKCUCX.TcTerminals210_EK1100_1.TcTerminals210_1BK1250.A_0331_KL_3214_4_Ch_ana_Input_PT100_RTD_3_wire.Channel_4.Data_Out <-> Channel 4/Data Out
//   PLC/PLC Instance <-> EtherCAT Master BKCUCX/TcTerminals210_EK1100_1/TcTerminals210_1BK1250/A_0333(KL 3222, 2 Ch. ana. Input PT100 (RTD, high-precision))
//     PlcTask Inputs/GVL_iXlinker.EtherCAT_Master_BKCUCX.TcTerminals210_EK1100_1.TcTerminals210_1BK1250.A_0333_KL_3222_2_Ch_ana_Input_PT100_RTD_high_precision.Channel_1.State <-> Channel 1/State
//     PlcTask Inputs/GVL_iXlinker.EtherCAT_Master_BKCUCX.TcTerminals210_EK1100_1.TcTerminals210_1BK1250.A_0333_KL_3222_2_Ch_ana_Input_PT100_RTD_high_precision.Channel_2.State <-> Channel 2/State
//     PlcTask Inputs/GVL_iXlinker.EtherCAT_Master_BKCUCX.TcTerminals210_EK1100_1.TcTerminals210_1BK1250.A_0333_KL_3222_2_Ch_ana_Input_PT100_RTD_high_precision.Channel_1.Data_In <-> Channel 1/Data In
//     PlcTask Inputs/GVL_iXlinker.EtherCAT_Master_BKCUCX.TcTerminals210_EK1100_1.TcTerminals210_1BK1250.A_0333_KL_3222_2_Ch_ana_Input_PT100_RTD_high_precision.Channel_2.Data_In <-> Channel 2/Data In
//     PlcTask Outputs/GVL_iXlinker.EtherCAT_Master_BKCUCX.TcTerminals210_EK1100_1.TcTerminals210_1BK1250.A_0333_KL_3222_2_Ch_ana_Input_PT100_RTD_high_precision.Channel_1.Ctrl <-> Channel 1/Ctrl
//     PlcTask Outputs/GVL_iXlinker.EtherCAT_Master_BKCUCX.TcTerminals210_EK1100_1.TcTerminals210_1BK1250.A_0333_KL_3222_2_Ch_ana_Input_PT100_RTD_high_precision.Channel_2.Ctrl <-> Channel 2/Ctrl
//     PlcTask Outputs/GVL_iXlinker.EtherCAT_Master_BKCUCX.TcTerminals210_EK1100_1.TcTerminals210_1BK1250.A_0333_KL_3222_2_Ch_ana_Input_PT100_RTD_high_precision.Channel_1.Data_Out <-> Channel 1/Data Out
//     PlcTask Outputs/GVL_iXlinker.EtherCAT_Master_BKCUCX.TcTerminals210_EK1100_1.TcTerminals210_1BK1250.A_0333_KL_3222_2_Ch_ana_Input_PT100_RTD_high_precision.Channel_2.Data_Out <-> Channel 2/Data Out
//   PLC/PLC Instance <-> EtherCAT Master BKCUCX/TcTerminals210_EK1100_1/TcTerminals210_1BK1250/A_0335(KL 3224)
//     PlcTask Inputs/GVL_iXlinker.EtherCAT_Master_BKCUCX.TcTerminals210_EK1100_1.TcTerminals210_1BK1250.A_0335_KL_3224.Channel_1.State <-> Channel 1/State
//     PlcTask Inputs/GVL_iXlinker.EtherCAT_Master_BKCUCX.TcTerminals210_EK1100_1.TcTerminals210_1BK1250.A_0335_KL_3224.Channel_2.State <-> Channel 2/State
//     PlcTask Inputs/GVL_iXlinker.EtherCAT_Master_BKCUCX.TcTerminals210_EK1100_1.TcTerminals210_1BK1250.A_0335_KL_3224.Channel_3.State <-> Channel 3/State
//     PlcTask Inputs/GVL_iXlinker.EtherCAT_Master_BKCUCX.TcTerminals210_EK1100_1.TcTerminals210_1BK1250.A_0335_KL_3224.Channel_4.State <-> Channel 4/State
//     PlcTask Inputs/GVL_iXlinker.EtherCAT_Master_BKCUCX.TcTerminals210_EK1100_1.TcTerminals210_1BK1250.A_0335_KL_3224.Channel_1.Data_In <-> Channel 1/Data In
//     PlcTask Inputs/GVL_iXlinker.EtherCAT_Master_BKCUCX.TcTerminals210_EK1100_1.TcTerminals210_1BK1250.A_0335_KL_3224.Channel_2.Data_In <-> Channel 2/Data In
//     PlcTask Inputs/GVL_iXlinker.EtherCAT_Master_BKCUCX.TcTerminals210_EK1100_1.TcTerminals210_1BK1250.A_0335_KL_3224.Channel_3.Data_In <-> Channel 3/Data In
//     PlcTask Inputs/GVL_iXlinker.EtherCAT_Master_BKCUCX.TcTerminals210_EK1100_1.TcTerminals210_1BK1250.A_0335_KL_3224.Channel_4.Data_In <-> Channel 4/Data In
//     PlcTask Outputs/GVL_iXlinker.EtherCAT_Master_BKCUCX.TcTerminals210_EK1100_1.TcTerminals210_1BK1250.A_0335_KL_3224.Channel_1.Ctrl <-> Channel 1/Ctrl
//     PlcTask Outputs/GVL_iXlinker.EtherCAT_Master_BKCUCX.TcTerminals210_EK1100_1.TcTerminals210_1BK1250.A_0335_KL_3224.Channel_2.Ctrl <-> Channel 2/Ctrl
//     PlcTask Outputs/GVL_iXlinker.EtherCAT_Master_BKCUCX.TcTerminals210_EK1100_1.TcTerminals210_1BK1250.A_0335_KL_3224.Channel_3.Ctrl <-> Channel 3/Ctrl
//     PlcTask Outputs/GVL_iXlinker.EtherCAT_Master_BKCUCX.TcTerminals210_EK1100_1.TcTerminals210_1BK1250.A_0335_KL_3224.Channel_4.Ctrl <-> Channel 4/Ctrl
//     PlcTask Outputs/GVL_iXlinker.EtherCAT_Master_BKCUCX.TcTerminals210_EK1100_1.TcTerminals210_1BK1250.A_0335_KL_3224.Channel_1.Data_Out <-> Channel 1/Data Out
//     PlcTask Outputs/GVL_iXlinker.EtherCAT_Master_BKCUCX.TcTerminals210_EK1100_1.TcTerminals210_1BK1250.A_0335_KL_3224.Channel_2.Data_Out <-> Channel 2/Data Out
//     PlcTask Outputs/GVL_iXlinker.EtherCAT_Master_BKCUCX.TcTerminals210_EK1100_1.TcTerminals210_1BK1250.A_0335_KL_3224.Channel_3.Data_Out <-> Channel 3/Data Out
//     PlcTask Outputs/GVL_iXlinker.EtherCAT_Master_BKCUCX.TcTerminals210_EK1100_1.TcTerminals210_1BK1250.A_0335_KL_3224.Channel_4.Data_Out <-> Channel 4/Data Out
//   PLC/PLC Instance <-> EtherCAT Master BKCUCX/TcTerminals210_EK1100_1/TcTerminals210_1BK1250/A_0337(KL 3228, 4 of 8 Ch. ana. Input PT1000, Ni1000 (RTD))
//     PlcTask Inputs/GVL_iXlinker.EtherCAT_Master_BKCUCX.TcTerminals210_EK1100_1.TcTerminals210_1BK1250.A_0337_KL_3228_4_of_8_Ch_ana_Input_PT1000_Ni1000_RTD.Channel_1.State <-> Channel 1/State
//     PlcTask Inputs/GVL_iXlinker.EtherCAT_Master_BKCUCX.TcTerminals210_EK1100_1.TcTerminals210_1BK1250.A_0337_KL_3228_4_of_8_Ch_ana_Input_PT1000_Ni1000_RTD.Channel_2.State <-> Channel 2/State
//     PlcTask Inputs/GVL_iXlinker.EtherCAT_Master_BKCUCX.TcTerminals210_EK1100_1.TcTerminals210_1BK1250.A_0337_KL_3228_4_of_8_Ch_ana_Input_PT1000_Ni1000_RTD.Channel_3.State <-> Channel 3/State
//     PlcTask Inputs/GVL_iXlinker.EtherCAT_Master_BKCUCX.TcTerminals210_EK1100_1.TcTerminals210_1BK1250.A_0337_KL_3228_4_of_8_Ch_ana_Input_PT1000_Ni1000_RTD.Channel_4.State <-> Channel 4/State
//     PlcTask Inputs/GVL_iXlinker.EtherCAT_Master_BKCUCX.TcTerminals210_EK1100_1.TcTerminals210_1BK1250.A_0337_KL_3228_4_of_8_Ch_ana_Input_PT1000_Ni1000_RTD.Channel_1.Data_In <-> Channel 1/Data In
//     PlcTask Inputs/GVL_iXlinker.EtherCAT_Master_BKCUCX.TcTerminals210_EK1100_1.TcTerminals210_1BK1250.A_0337_KL_3228_4_of_8_Ch_ana_Input_PT1000_Ni1000_RTD.Channel_2.Data_In <-> Channel 2/Data In
//     PlcTask Inputs/GVL_iXlinker.EtherCAT_Master_BKCUCX.TcTerminals210_EK1100_1.TcTerminals210_1BK1250.A_0337_KL_3228_4_of_8_Ch_ana_Input_PT1000_Ni1000_RTD.Channel_3.Data_In <-> Channel 3/Data In
//     PlcTask Inputs/GVL_iXlinker.EtherCAT_Master_BKCUCX.TcTerminals210_EK1100_1.TcTerminals210_1BK1250.A_0337_KL_3228_4_of_8_Ch_ana_Input_PT1000_Ni1000_RTD.Channel_4.Data_In <-> Channel 4/Data In
//     PlcTask Outputs/GVL_iXlinker.EtherCAT_Master_BKCUCX.TcTerminals210_EK1100_1.TcTerminals210_1BK1250.A_0337_KL_3228_4_of_8_Ch_ana_Input_PT1000_Ni1000_RTD.Channel_1.Ctrl <-> Channel 1/Ctrl
//     PlcTask Outputs/GVL_iXlinker.EtherCAT_Master_BKCUCX.TcTerminals210_EK1100_1.TcTerminals210_1BK1250.A_0337_KL_3228_4_of_8_Ch_ana_Input_PT1000_Ni1000_RTD.Channel_2.Ctrl <-> Channel 2/Ctrl
//     PlcTask Outputs/GVL_iXlinker.EtherCAT_Master_BKCUCX.TcTerminals210_EK1100_1.TcTerminals210_1BK1250.A_0337_KL_3228_4_of_8_Ch_ana_Input_PT1000_Ni1000_RTD.Channel_3.Ctrl <-> Channel 3/Ctrl
//     PlcTask Outputs/GVL_iXlinker.EtherCAT_Master_BKCUCX.TcTerminals210_EK1100_1.TcTerminals210_1BK1250.A_0337_KL_3228_4_of_8_Ch_ana_Input_PT1000_Ni1000_RTD.Channel_4.Ctrl <-> Channel 4/Ctrl
//     PlcTask Outputs/GVL_iXlinker.EtherCAT_Master_BKCUCX.TcTerminals210_EK1100_1.TcTerminals210_1BK1250.A_0337_KL_3228_4_of_8_Ch_ana_Input_PT1000_Ni1000_RTD.Channel_1.Data_Out <-> Channel 1/Data Out
//     PlcTask Outputs/GVL_iXlinker.EtherCAT_Master_BKCUCX.TcTerminals210_EK1100_1.TcTerminals210_1BK1250.A_0337_KL_3228_4_of_8_Ch_ana_Input_PT1000_Ni1000_RTD.Channel_2.Data_Out <-> Channel 2/Data Out
//     PlcTask Outputs/GVL_iXlinker.EtherCAT_Master_BKCUCX.TcTerminals210_EK1100_1.TcTerminals210_1BK1250.A_0337_KL_3228_4_of_8_Ch_ana_Input_PT1000_Ni1000_RTD.Channel_3.Data_Out <-> Channel 3/Data Out
//     PlcTask Outputs/GVL_iXlinker.EtherCAT_Master_BKCUCX.TcTerminals210_EK1100_1.TcTerminals210_1BK1250.A_0337_KL_3228_4_of_8_Ch_ana_Input_PT1000_Ni1000_RTD.Channel_4.Data_Out <-> Channel 4/Data Out
//   PLC/PLC Instance <-> EtherCAT Master BKCUCX/TcTerminals210_EK1100_1/TcTerminals210_1BK1250/A_0339(KL 3302, 2 Ch. ana. Input Thermo)
//     PlcTask Inputs/GVL_iXlinker.EtherCAT_Master_BKCUCX.TcTerminals210_EK1100_1.TcTerminals210_1BK1250.A_0339_KL_3302_2_Ch_ana_Input_Thermo.Channel_1.State <-> Channel 1/State
//     PlcTask Inputs/GVL_iXlinker.EtherCAT_Master_BKCUCX.TcTerminals210_EK1100_1.TcTerminals210_1BK1250.A_0339_KL_3302_2_Ch_ana_Input_Thermo.Channel_2.State <-> Channel 2/State
//     PlcTask Inputs/GVL_iXlinker.EtherCAT_Master_BKCUCX.TcTerminals210_EK1100_1.TcTerminals210_1BK1250.A_0339_KL_3302_2_Ch_ana_Input_Thermo.Channel_1.Data_In <-> Channel 1/Data In
//     PlcTask Inputs/GVL_iXlinker.EtherCAT_Master_BKCUCX.TcTerminals210_EK1100_1.TcTerminals210_1BK1250.A_0339_KL_3302_2_Ch_ana_Input_Thermo.Channel_2.Data_In <-> Channel 2/Data In
//     PlcTask Outputs/GVL_iXlinker.EtherCAT_Master_BKCUCX.TcTerminals210_EK1100_1.TcTerminals210_1BK1250.A_0339_KL_3302_2_Ch_ana_Input_Thermo.Channel_1.Ctrl <-> Channel 1/Ctrl
//     PlcTask Outputs/GVL_iXlinker.EtherCAT_Master_BKCUCX.TcTerminals210_EK1100_1.TcTerminals210_1BK1250.A_0339_KL_3302_2_Ch_ana_Input_Thermo.Channel_2.Ctrl <-> Channel 2/Ctrl
//     PlcTask Outputs/GVL_iXlinker.EtherCAT_Master_BKCUCX.TcTerminals210_EK1100_1.TcTerminals210_1BK1250.A_0339_KL_3302_2_Ch_ana_Input_Thermo.Channel_1.Data_Out <-> Channel 1/Data Out
//     PlcTask Outputs/GVL_iXlinker.EtherCAT_Master_BKCUCX.TcTerminals210_EK1100_1.TcTerminals210_1BK1250.A_0339_KL_3302_2_Ch_ana_Input_Thermo.Channel_2.Data_Out <-> Channel 2/Data Out
//   PLC/PLC Instance <-> EtherCAT Master BKCUCX/TcTerminals210_EK1100_1/TcTerminals210_1BK1250/A_0341(KL 3311, 1 Ch. ana. Input Thermo with wire break recog.)
//     PlcTask Inputs/GVL_iXlinker.EtherCAT_Master_BKCUCX.TcTerminals210_EK1100_1.TcTerminals210_1BK1250.A_0341_KL_3311_1_Ch_ana_Input_Thermo_with_wire_break_recog.Channel_1.State <-> Channel 1/State
//     PlcTask Inputs/GVL_iXlinker.EtherCAT_Master_BKCUCX.TcTerminals210_EK1100_1.TcTerminals210_1BK1250.A_0341_KL_3311_1_Ch_ana_Input_Thermo_with_wire_break_recog.Channel_1.Data_In <-> Channel 1/Data In
//     PlcTask Outputs/GVL_iXlinker.EtherCAT_Master_BKCUCX.TcTerminals210_EK1100_1.TcTerminals210_1BK1250.A_0341_KL_3311_1_Ch_ana_Input_Thermo_with_wire_break_recog.Channel_1.Ctrl <-> Channel 1/Ctrl
//     PlcTask Outputs/GVL_iXlinker.EtherCAT_Master_BKCUCX.TcTerminals210_EK1100_1.TcTerminals210_1BK1250.A_0341_KL_3311_1_Ch_ana_Input_Thermo_with_wire_break_recog.Channel_1.Data_Out <-> Channel 1/Data Out
//   PLC/PLC Instance <-> EtherCAT Master BKCUCX/TcTerminals210_EK1100_1/TcTerminals210_1BK1250/A_0343(KL 3312, 2 Ch. ana. Input Thermo with wire break recog.)
//     PlcTask Inputs/GVL_iXlinker.EtherCAT_Master_BKCUCX.TcTerminals210_EK1100_1.TcTerminals210_1BK1250.A_0343_KL_3312_2_Ch_ana_Input_Thermo_with_wire_break_recog.Channel_1.State <-> Channel 1/State
//     PlcTask Inputs/GVL_iXlinker.EtherCAT_Master_BKCUCX.TcTerminals210_EK1100_1.TcTerminals210_1BK1250.A_0343_KL_3312_2_Ch_ana_Input_Thermo_with_wire_break_recog.Channel_2.State <-> Channel 2/State
//     PlcTask Inputs/GVL_iXlinker.EtherCAT_Master_BKCUCX.TcTerminals210_EK1100_1.TcTerminals210_1BK1250.A_0343_KL_3312_2_Ch_ana_Input_Thermo_with_wire_break_recog.Channel_1.Data_In <-> Channel 1/Data In
//     PlcTask Inputs/GVL_iXlinker.EtherCAT_Master_BKCUCX.TcTerminals210_EK1100_1.TcTerminals210_1BK1250.A_0343_KL_3312_2_Ch_ana_Input_Thermo_with_wire_break_recog.Channel_2.Data_In <-> Channel 2/Data In
//     PlcTask Outputs/GVL_iXlinker.EtherCAT_Master_BKCUCX.TcTerminals210_EK1100_1.TcTerminals210_1BK1250.A_0343_KL_3312_2_Ch_ana_Input_Thermo_with_wire_break_recog.Channel_1.Ctrl <-> Channel 1/Ctrl
//     PlcTask Outputs/GVL_iXlinker.EtherCAT_Master_BKCUCX.TcTerminals210_EK1100_1.TcTerminals210_1BK1250.A_0343_KL_3312_2_Ch_ana_Input_Thermo_with_wire_break_recog.Channel_2.Ctrl <-> Channel 2/Ctrl
//     PlcTask Outputs/GVL_iXlinker.EtherCAT_Master_BKCUCX.TcTerminals210_EK1100_1.TcTerminals210_1BK1250.A_0343_KL_3312_2_Ch_ana_Input_Thermo_with_wire_break_recog.Channel_1.Data_Out <-> Channel 1/Data Out
//     PlcTask Outputs/GVL_iXlinker.EtherCAT_Master_BKCUCX.TcTerminals210_EK1100_1.TcTerminals210_1BK1250.A_0343_KL_3312_2_Ch_ana_Input_Thermo_with_wire_break_recog.Channel_2.Data_Out <-> Channel 2/Data Out
//   PLC/PLC Instance <-> EtherCAT Master BKCUCX/TcTerminals210_EK1100_1/TcTerminals210_1BK1250/A_0345(KL 3314, 4 Ch. ana. Input Thermo with wire break recog.)
//     PlcTask Inputs/GVL_iXlinker.EtherCAT_Master_BKCUCX.TcTerminals210_EK1100_1.TcTerminals210_1BK1250.A_0345_KL_3314_4_Ch_ana_Input_Thermo_with_wire_break_recog.Channel_1.State <-> Channel 1/State
//     PlcTask Inputs/GVL_iXlinker.EtherCAT_Master_BKCUCX.TcTerminals210_EK1100_1.TcTerminals210_1BK1250.A_0345_KL_3314_4_Ch_ana_Input_Thermo_with_wire_break_recog.Channel_2.State <-> Channel 2/State
//     PlcTask Inputs/GVL_iXlinker.EtherCAT_Master_BKCUCX.TcTerminals210_EK1100_1.TcTerminals210_1BK1250.A_0345_KL_3314_4_Ch_ana_Input_Thermo_with_wire_break_recog.Channel_3.State <-> Channel 3/State
//     PlcTask Inputs/GVL_iXlinker.EtherCAT_Master_BKCUCX.TcTerminals210_EK1100_1.TcTerminals210_1BK1250.A_0345_KL_3314_4_Ch_ana_Input_Thermo_with_wire_break_recog.Channel_4.State <-> Channel 4/State
//     PlcTask Inputs/GVL_iXlinker.EtherCAT_Master_BKCUCX.TcTerminals210_EK1100_1.TcTerminals210_1BK1250.A_0345_KL_3314_4_Ch_ana_Input_Thermo_with_wire_break_recog.Channel_1.Data_In <-> Channel 1/Data In
//     PlcTask Inputs/GVL_iXlinker.EtherCAT_Master_BKCUCX.TcTerminals210_EK1100_1.TcTerminals210_1BK1250.A_0345_KL_3314_4_Ch_ana_Input_Thermo_with_wire_break_recog.Channel_2.Data_In <-> Channel 2/Data In
//     PlcTask Inputs/GVL_iXlinker.EtherCAT_Master_BKCUCX.TcTerminals210_EK1100_1.TcTerminals210_1BK1250.A_0345_KL_3314_4_Ch_ana_Input_Thermo_with_wire_break_recog.Channel_3.Data_In <-> Channel 3/Data In
//     PlcTask Inputs/GVL_iXlinker.EtherCAT_Master_BKCUCX.TcTerminals210_EK1100_1.TcTerminals210_1BK1250.A_0345_KL_3314_4_Ch_ana_Input_Thermo_with_wire_break_recog.Channel_4.Data_In <-> Channel 4/Data In
//     PlcTask Outputs/GVL_iXlinker.EtherCAT_Master_BKCUCX.TcTerminals210_EK1100_1.TcTerminals210_1BK1250.A_0345_KL_3314_4_Ch_ana_Input_Thermo_with_wire_break_recog.Channel_1.Ctrl <-> Channel 1/Ctrl
//     PlcTask Outputs/GVL_iXlinker.EtherCAT_Master_BKCUCX.TcTerminals210_EK1100_1.TcTerminals210_1BK1250.A_0345_KL_3314_4_Ch_ana_Input_Thermo_with_wire_break_recog.Channel_2.Ctrl <-> Channel 2/Ctrl
//     PlcTask Outputs/GVL_iXlinker.EtherCAT_Master_BKCUCX.TcTerminals210_EK1100_1.TcTerminals210_1BK1250.A_0345_KL_3314_4_Ch_ana_Input_Thermo_with_wire_break_recog.Channel_3.Ctrl <-> Channel 3/Ctrl
//     PlcTask Outputs/GVL_iXlinker.EtherCAT_Master_BKCUCX.TcTerminals210_EK1100_1.TcTerminals210_1BK1250.A_0345_KL_3314_4_Ch_ana_Input_Thermo_with_wire_break_recog.Channel_4.Ctrl <-> Channel 4/Ctrl
//     PlcTask Outputs/GVL_iXlinker.EtherCAT_Master_BKCUCX.TcTerminals210_EK1100_1.TcTerminals210_1BK1250.A_0345_KL_3314_4_Ch_ana_Input_Thermo_with_wire_break_recog.Channel_1.Data_Out <-> Channel 1/Data Out
//     PlcTask Outputs/GVL_iXlinker.EtherCAT_Master_BKCUCX.TcTerminals210_EK1100_1.TcTerminals210_1BK1250.A_0345_KL_3314_4_Ch_ana_Input_Thermo_with_wire_break_recog.Channel_2.Data_Out <-> Channel 2/Data Out
//     PlcTask Outputs/GVL_iXlinker.EtherCAT_Master_BKCUCX.TcTerminals210_EK1100_1.TcTerminals210_1BK1250.A_0345_KL_3314_4_Ch_ana_Input_Thermo_with_wire_break_recog.Channel_3.Data_Out <-> Channel 3/Data Out
//     PlcTask Outputs/GVL_iXlinker.EtherCAT_Master_BKCUCX.TcTerminals210_EK1100_1.TcTerminals210_1BK1250.A_0345_KL_3314_4_Ch_ana_Input_Thermo_with_wire_break_recog.Channel_4.Data_Out <-> Channel 4/Data Out
//   PLC/PLC Instance <-> EtherCAT Master BKCUCX/TcTerminals210_EK1100_1/TcTerminals210_1BK1250/A_0347(KL 3351, 1 Ch. Resistor Bridge)
//     PlcTask Inputs/GVL_iXlinker.EtherCAT_Master_BKCUCX.TcTerminals210_EK1100_1.TcTerminals210_1BK1250.A_0347_KL_3351_1_Ch_Resistor_Bridge.Channel_1.Status <-> Channel 1/Status
//     PlcTask Inputs/GVL_iXlinker.EtherCAT_Master_BKCUCX.TcTerminals210_EK1100_1.TcTerminals210_1BK1250.A_0347_KL_3351_1_Ch_Resistor_Bridge.Channel_1.Ud_RegIn <-> Channel 1/Ud_RegIn
//     PlcTask Inputs/GVL_iXlinker.EtherCAT_Master_BKCUCX.TcTerminals210_EK1100_1.TcTerminals210_1BK1250.A_0347_KL_3351_1_Ch_Resistor_Bridge.Channel_1.Uref <-> Channel 1/Uref
//     PlcTask Outputs/GVL_iXlinker.EtherCAT_Master_BKCUCX.TcTerminals210_EK1100_1.TcTerminals210_1BK1250.A_0347_KL_3351_1_Ch_Resistor_Bridge.Channel_1.Ctrl <-> Channel 1/Ctrl
//     PlcTask Outputs/GVL_iXlinker.EtherCAT_Master_BKCUCX.TcTerminals210_EK1100_1.TcTerminals210_1BK1250.A_0347_KL_3351_1_Ch_Resistor_Bridge.Channel_1.RegOut <-> Channel 1/RegOut
//   PLC/PLC Instance <-> EtherCAT Master BKCUCX/TcTerminals210_EK1100_1/TcTerminals210_1BK1250/A_0350(KL 3351-0001, 1 Ch. Resistor Bridge)
//     PlcTask Inputs/GVL_iXlinker.EtherCAT_Master_BKCUCX.TcTerminals210_EK1100_1.TcTerminals210_1BK1250.A_0350_KL_3351_0001_1_Ch_Resistor_Bridge.Channel_1.Status <-> Channel 1/Status
//     PlcTask Inputs/GVL_iXlinker.EtherCAT_Master_BKCUCX.TcTerminals210_EK1100_1.TcTerminals210_1BK1250.A_0350_KL_3351_0001_1_Ch_Resistor_Bridge.Channel_1.Ud_RegIn <-> Channel 1/Ud_RegIn
//     PlcTask Inputs/GVL_iXlinker.EtherCAT_Master_BKCUCX.TcTerminals210_EK1100_1.TcTerminals210_1BK1250.A_0350_KL_3351_0001_1_Ch_Resistor_Bridge.Channel_1.Uref <-> Channel 1/Uref
//     PlcTask Outputs/GVL_iXlinker.EtherCAT_Master_BKCUCX.TcTerminals210_EK1100_1.TcTerminals210_1BK1250.A_0350_KL_3351_0001_1_Ch_Resistor_Bridge.Channel_1.Ctrl <-> Channel 1/Ctrl
//     PlcTask Outputs/GVL_iXlinker.EtherCAT_Master_BKCUCX.TcTerminals210_EK1100_1.TcTerminals210_1BK1250.A_0350_KL_3351_0001_1_Ch_Resistor_Bridge.Channel_1.RegOut <-> Channel 1/RegOut
//     PlcTask Outputs/GVL_iXlinker.EtherCAT_Master_BKCUCX.TcTerminals210_EK1100_1.TcTerminals210_1BK1250.A_0350_KL_3351_0001_1_Ch_Resistor_Bridge.Channel_1.Ctrl1 <-> Channel 1/Ctrl1
//   PLC/PLC Instance <-> EtherCAT Master BKCUCX/TcTerminals210_EK1100_1/TcTerminals210_1BK1250/A_0353(KL 3356, 1 Ch. precise Resistor Bridge)
//     PlcTask Inputs/GVL_iXlinker.EtherCAT_Master_BKCUCX.TcTerminals210_EK1100_1.TcTerminals210_1BK1250.A_0353_KL_3356_1_Ch_precise_Resistor_Bridge.Channel_1.Status <-> Channel 1/Status
//     PlcTask Inputs/GVL_iXlinker.EtherCAT_Master_BKCUCX.TcTerminals210_EK1100_1.TcTerminals210_1BK1250.A_0353_KL_3356_1_Ch_precise_Resistor_Bridge.Channel_1.RegIn <-> Channel 1/RegIn
//     PlcTask Inputs/GVL_iXlinker.EtherCAT_Master_BKCUCX.TcTerminals210_EK1100_1.TcTerminals210_1BK1250.A_0353_KL_3356_1_Ch_precise_Resistor_Bridge.Channel_1.AnStatus <-> Channel 1/AnStatus
//     PlcTask Inputs/GVL_iXlinker.EtherCAT_Master_BKCUCX.TcTerminals210_EK1100_1.TcTerminals210_1BK1250.A_0353_KL_3356_1_Ch_precise_Resistor_Bridge.Channel_1.Weight <-> Channel 1/Weight
//     PlcTask Outputs/GVL_iXlinker.EtherCAT_Master_BKCUCX.TcTerminals210_EK1100_1.TcTerminals210_1BK1250.A_0353_KL_3356_1_Ch_precise_Resistor_Bridge.Channel_1.Ctrl <-> Channel 1/Ctrl
//     PlcTask Outputs/GVL_iXlinker.EtherCAT_Master_BKCUCX.TcTerminals210_EK1100_1.TcTerminals210_1BK1250.A_0353_KL_3356_1_Ch_precise_Resistor_Bridge.Channel_1.RegOut <-> Channel 1/RegOut
//     PlcTask Outputs/GVL_iXlinker.EtherCAT_Master_BKCUCX.TcTerminals210_EK1100_1.TcTerminals210_1BK1250.A_0353_KL_3356_1_Ch_precise_Resistor_Bridge.Channel_1.AnCtrl <-> Channel 1/AnCtrl
//   PLC/PLC Instance <-> EtherCAT Master BKCUCX/TcTerminals210_EK1100_1/TcTerminals210_1BK1250/A_0356(KL 3361, 1 Ch. Oscilloscope)
//     PlcTask Inputs/GVL_iXlinker.EtherCAT_Master_BKCUCX.TcTerminals210_EK1100_1.TcTerminals210_1BK1250.A_0356_KL_3361_1_Ch_Oscilloscope.Channel_1.State <-> Channel 1/State
//     PlcTask Inputs/GVL_iXlinker.EtherCAT_Master_BKCUCX.TcTerminals210_EK1100_1.TcTerminals210_1BK1250.A_0356_KL_3361_1_Ch_Oscilloscope.Channel_1.Data_In <-> Channel 1/Data In
//     PlcTask Outputs/GVL_iXlinker.EtherCAT_Master_BKCUCX.TcTerminals210_EK1100_1.TcTerminals210_1BK1250.A_0356_KL_3361_1_Ch_Oscilloscope.Channel_1.Ctrl <-> Channel 1/Ctrl
//     PlcTask Outputs/GVL_iXlinker.EtherCAT_Master_BKCUCX.TcTerminals210_EK1100_1.TcTerminals210_1BK1250.A_0356_KL_3361_1_Ch_Oscilloscope.Channel_1.Data_Out <-> Channel 1/Data Out
//   PLC/PLC Instance <-> EtherCAT Master BKCUCX/TcTerminals210_EK1100_1/TcTerminals210_1BK1250/A_0358(KL 3361-1001, 1 Ch. Oscilloscope)
//     PlcTask Inputs/GVL_iXlinker.EtherCAT_Master_BKCUCX.TcTerminals210_EK1100_1.TcTerminals210_1BK1250.A_0358_KL_3361_1001_1_Ch_Oscilloscope.Channel_1.State <-> Channel 1/State
//     PlcTask Inputs/GVL_iXlinker.EtherCAT_Master_BKCUCX.TcTerminals210_EK1100_1.TcTerminals210_1BK1250.A_0358_KL_3361_1001_1_Ch_Oscilloscope.Channel_1.Data_In_0 <-> Channel 1/Data In 0
//     PlcTask Inputs/GVL_iXlinker.EtherCAT_Master_BKCUCX.TcTerminals210_EK1100_1.TcTerminals210_1BK1250.A_0358_KL_3361_1001_1_Ch_Oscilloscope.Channel_1.Data_In_1 <-> Channel 1/Data In 1
//     PlcTask Inputs/GVL_iXlinker.EtherCAT_Master_BKCUCX.TcTerminals210_EK1100_1.TcTerminals210_1BK1250.A_0358_KL_3361_1001_1_Ch_Oscilloscope.Channel_1.Data_In_2 <-> Channel 1/Data In 2
//     PlcTask Inputs/GVL_iXlinker.EtherCAT_Master_BKCUCX.TcTerminals210_EK1100_1.TcTerminals210_1BK1250.A_0358_KL_3361_1001_1_Ch_Oscilloscope.Channel_1.Data_In_3 <-> Channel 1/Data In 3
//     PlcTask Inputs/GVL_iXlinker.EtherCAT_Master_BKCUCX.TcTerminals210_EK1100_1.TcTerminals210_1BK1250.A_0358_KL_3361_1001_1_Ch_Oscilloscope.Channel_1.Data_In_4 <-> Channel 1/Data In 4
//     PlcTask Inputs/GVL_iXlinker.EtherCAT_Master_BKCUCX.TcTerminals210_EK1100_1.TcTerminals210_1BK1250.A_0358_KL_3361_1001_1_Ch_Oscilloscope.Channel_1.Data_In_5 <-> Channel 1/Data In 5
//     PlcTask Inputs/GVL_iXlinker.EtherCAT_Master_BKCUCX.TcTerminals210_EK1100_1.TcTerminals210_1BK1250.A_0358_KL_3361_1001_1_Ch_Oscilloscope.Channel_1.Data_In_6 <-> Channel 1/Data In 6
//     PlcTask Inputs/GVL_iXlinker.EtherCAT_Master_BKCUCX.TcTerminals210_EK1100_1.TcTerminals210_1BK1250.A_0358_KL_3361_1001_1_Ch_Oscilloscope.Channel_1.Data_In_7 <-> Channel 1/Data In 7
//     PlcTask Inputs/GVL_iXlinker.EtherCAT_Master_BKCUCX.TcTerminals210_EK1100_1.TcTerminals210_1BK1250.A_0358_KL_3361_1001_1_Ch_Oscilloscope.Channel_1.Data_In_8 <-> Channel 1/Data In 8
//     PlcTask Inputs/GVL_iXlinker.EtherCAT_Master_BKCUCX.TcTerminals210_EK1100_1.TcTerminals210_1BK1250.A_0358_KL_3361_1001_1_Ch_Oscilloscope.Channel_1.Data_In_9 <-> Channel 1/Data In 9
//     PlcTask Inputs/GVL_iXlinker.EtherCAT_Master_BKCUCX.TcTerminals210_EK1100_1.TcTerminals210_1BK1250.A_0358_KL_3361_1001_1_Ch_Oscilloscope.Channel_1.Data_In_10 <-> Channel 1/Data In 10
//     PlcTask Outputs/GVL_iXlinker.EtherCAT_Master_BKCUCX.TcTerminals210_EK1100_1.TcTerminals210_1BK1250.A_0358_KL_3361_1001_1_Ch_Oscilloscope.Channel_1.Ctrl <-> Channel 1/Ctrl
//     PlcTask Outputs/GVL_iXlinker.EtherCAT_Master_BKCUCX.TcTerminals210_EK1100_1.TcTerminals210_1BK1250.A_0358_KL_3361_1001_1_Ch_Oscilloscope.Channel_1.Data_Out_0 <-> Channel 1/Data Out 0
//     PlcTask Outputs/GVL_iXlinker.EtherCAT_Master_BKCUCX.TcTerminals210_EK1100_1.TcTerminals210_1BK1250.A_0358_KL_3361_1001_1_Ch_Oscilloscope.Channel_1.Data_Out_1 <-> Channel 1/Data Out 1
//     PlcTask Outputs/GVL_iXlinker.EtherCAT_Master_BKCUCX.TcTerminals210_EK1100_1.TcTerminals210_1BK1250.A_0358_KL_3361_1001_1_Ch_Oscilloscope.Channel_1.Data_Out_2 <-> Channel 1/Data Out 2
//     PlcTask Outputs/GVL_iXlinker.EtherCAT_Master_BKCUCX.TcTerminals210_EK1100_1.TcTerminals210_1BK1250.A_0358_KL_3361_1001_1_Ch_Oscilloscope.Channel_1.Data_Out_3 <-> Channel 1/Data Out 3
//     PlcTask Outputs/GVL_iXlinker.EtherCAT_Master_BKCUCX.TcTerminals210_EK1100_1.TcTerminals210_1BK1250.A_0358_KL_3361_1001_1_Ch_Oscilloscope.Channel_1.Data_Out_4 <-> Channel 1/Data Out 4
//     PlcTask Outputs/GVL_iXlinker.EtherCAT_Master_BKCUCX.TcTerminals210_EK1100_1.TcTerminals210_1BK1250.A_0358_KL_3361_1001_1_Ch_Oscilloscope.Channel_1.Data_Out_5 <-> Channel 1/Data Out 5
//     PlcTask Outputs/GVL_iXlinker.EtherCAT_Master_BKCUCX.TcTerminals210_EK1100_1.TcTerminals210_1BK1250.A_0358_KL_3361_1001_1_Ch_Oscilloscope.Channel_1.Data_Out_6 <-> Channel 1/Data Out 6
//     PlcTask Outputs/GVL_iXlinker.EtherCAT_Master_BKCUCX.TcTerminals210_EK1100_1.TcTerminals210_1BK1250.A_0358_KL_3361_1001_1_Ch_Oscilloscope.Channel_1.Data_Out_7 <-> Channel 1/Data Out 7
//     PlcTask Outputs/GVL_iXlinker.EtherCAT_Master_BKCUCX.TcTerminals210_EK1100_1.TcTerminals210_1BK1250.A_0358_KL_3361_1001_1_Ch_Oscilloscope.Channel_1.Data_Out_8 <-> Channel 1/Data Out 8
//     PlcTask Outputs/GVL_iXlinker.EtherCAT_Master_BKCUCX.TcTerminals210_EK1100_1.TcTerminals210_1BK1250.A_0358_KL_3361_1001_1_Ch_Oscilloscope.Channel_1.Data_Out_9 <-> Channel 1/Data Out 9
//     PlcTask Outputs/GVL_iXlinker.EtherCAT_Master_BKCUCX.TcTerminals210_EK1100_1.TcTerminals210_1BK1250.A_0358_KL_3361_1001_1_Ch_Oscilloscope.Channel_1.Data_Out_10 <-> Channel 1/Data Out 10
//   PLC/PLC Instance <-> EtherCAT Master BKCUCX/TcTerminals210_EK1100_1/TcTerminals210_1BK1250/A_0359(KL 3361-1002, 1 Ch. Oscilloscope)
//     PlcTask Inputs/GVL_iXlinker.EtherCAT_Master_BKCUCX.TcTerminals210_EK1100_1.TcTerminals210_1BK1250.A_0359_KL_3361_1002_1_Ch_Oscilloscope.Channel_1.State <-> Channel 1/State
//     PlcTask Inputs/GVL_iXlinker.EtherCAT_Master_BKCUCX.TcTerminals210_EK1100_1.TcTerminals210_1BK1250.A_0359_KL_3361_1002_1_Ch_Oscilloscope.Channel_1.Data_In_0 <-> Channel 1/Data In 0
//     PlcTask Inputs/GVL_iXlinker.EtherCAT_Master_BKCUCX.TcTerminals210_EK1100_1.TcTerminals210_1BK1250.A_0359_KL_3361_1002_1_Ch_Oscilloscope.Channel_1.Data_In_1 <-> Channel 1/Data In 1
//     PlcTask Inputs/GVL_iXlinker.EtherCAT_Master_BKCUCX.TcTerminals210_EK1100_1.TcTerminals210_1BK1250.A_0359_KL_3361_1002_1_Ch_Oscilloscope.Channel_1.Data_In_2 <-> Channel 1/Data In 2
//     PlcTask Inputs/GVL_iXlinker.EtherCAT_Master_BKCUCX.TcTerminals210_EK1100_1.TcTerminals210_1BK1250.A_0359_KL_3361_1002_1_Ch_Oscilloscope.Channel_1.Data_In_3 <-> Channel 1/Data In 3
//     PlcTask Inputs/GVL_iXlinker.EtherCAT_Master_BKCUCX.TcTerminals210_EK1100_1.TcTerminals210_1BK1250.A_0359_KL_3361_1002_1_Ch_Oscilloscope.Channel_1.Data_In_4 <-> Channel 1/Data In 4
//     PlcTask Inputs/GVL_iXlinker.EtherCAT_Master_BKCUCX.TcTerminals210_EK1100_1.TcTerminals210_1BK1250.A_0359_KL_3361_1002_1_Ch_Oscilloscope.Channel_1.Data_In_5 <-> Channel 1/Data In 5
//     PlcTask Inputs/GVL_iXlinker.EtherCAT_Master_BKCUCX.TcTerminals210_EK1100_1.TcTerminals210_1BK1250.A_0359_KL_3361_1002_1_Ch_Oscilloscope.Channel_1.Data_In_6 <-> Channel 1/Data In 6
//     PlcTask Inputs/GVL_iXlinker.EtherCAT_Master_BKCUCX.TcTerminals210_EK1100_1.TcTerminals210_1BK1250.A_0359_KL_3361_1002_1_Ch_Oscilloscope.Channel_1.Data_In_7 <-> Channel 1/Data In 7
//     PlcTask Inputs/GVL_iXlinker.EtherCAT_Master_BKCUCX.TcTerminals210_EK1100_1.TcTerminals210_1BK1250.A_0359_KL_3361_1002_1_Ch_Oscilloscope.Channel_1.Data_In_8 <-> Channel 1/Data In 8
//     PlcTask Inputs/GVL_iXlinker.EtherCAT_Master_BKCUCX.TcTerminals210_EK1100_1.TcTerminals210_1BK1250.A_0359_KL_3361_1002_1_Ch_Oscilloscope.Channel_1.Data_In_9 <-> Channel 1/Data In 9
//     PlcTask Inputs/GVL_iXlinker.EtherCAT_Master_BKCUCX.TcTerminals210_EK1100_1.TcTerminals210_1BK1250.A_0359_KL_3361_1002_1_Ch_Oscilloscope.Channel_1.Data_In_10 <-> Channel 1/Data In 10
//     PlcTask Outputs/GVL_iXlinker.EtherCAT_Master_BKCUCX.TcTerminals210_EK1100_1.TcTerminals210_1BK1250.A_0359_KL_3361_1002_1_Ch_Oscilloscope.Channel_1.Ctrl <-> Channel 1/Ctrl
//     PlcTask Outputs/GVL_iXlinker.EtherCAT_Master_BKCUCX.TcTerminals210_EK1100_1.TcTerminals210_1BK1250.A_0359_KL_3361_1002_1_Ch_Oscilloscope.Channel_1.Data_Out_0 <-> Channel 1/Data Out 0
//     PlcTask Outputs/GVL_iXlinker.EtherCAT_Master_BKCUCX.TcTerminals210_EK1100_1.TcTerminals210_1BK1250.A_0359_KL_3361_1002_1_Ch_Oscilloscope.Channel_1.Data_Out_1 <-> Channel 1/Data Out 1
//     PlcTask Outputs/GVL_iXlinker.EtherCAT_Master_BKCUCX.TcTerminals210_EK1100_1.TcTerminals210_1BK1250.A_0359_KL_3361_1002_1_Ch_Oscilloscope.Channel_1.Data_Out_2 <-> Channel 1/Data Out 2
//     PlcTask Outputs/GVL_iXlinker.EtherCAT_Master_BKCUCX.TcTerminals210_EK1100_1.TcTerminals210_1BK1250.A_0359_KL_3361_1002_1_Ch_Oscilloscope.Channel_1.Data_Out_3 <-> Channel 1/Data Out 3
//     PlcTask Outputs/GVL_iXlinker.EtherCAT_Master_BKCUCX.TcTerminals210_EK1100_1.TcTerminals210_1BK1250.A_0359_KL_3361_1002_1_Ch_Oscilloscope.Channel_1.Data_Out_4 <-> Channel 1/Data Out 4
//     PlcTask Outputs/GVL_iXlinker.EtherCAT_Master_BKCUCX.TcTerminals210_EK1100_1.TcTerminals210_1BK1250.A_0359_KL_3361_1002_1_Ch_Oscilloscope.Channel_1.Data_Out_5 <-> Channel 1/Data Out 5
//     PlcTask Outputs/GVL_iXlinker.EtherCAT_Master_BKCUCX.TcTerminals210_EK1100_1.TcTerminals210_1BK1250.A_0359_KL_3361_1002_1_Ch_Oscilloscope.Channel_1.Data_Out_6 <-> Channel 1/Data Out 6
//     PlcTask Outputs/GVL_iXlinker.EtherCAT_Master_BKCUCX.TcTerminals210_EK1100_1.TcTerminals210_1BK1250.A_0359_KL_3361_1002_1_Ch_Oscilloscope.Channel_1.Data_Out_7 <-> Channel 1/Data Out 7
//     PlcTask Outputs/GVL_iXlinker.EtherCAT_Master_BKCUCX.TcTerminals210_EK1100_1.TcTerminals210_1BK1250.A_0359_KL_3361_1002_1_Ch_Oscilloscope.Channel_1.Data_Out_8 <-> Channel 1/Data Out 8
//     PlcTask Outputs/GVL_iXlinker.EtherCAT_Master_BKCUCX.TcTerminals210_EK1100_1.TcTerminals210_1BK1250.A_0359_KL_3361_1002_1_Ch_Oscilloscope.Channel_1.Data_Out_9 <-> Channel 1/Data Out 9
//     PlcTask Outputs/GVL_iXlinker.EtherCAT_Master_BKCUCX.TcTerminals210_EK1100_1.TcTerminals210_1BK1250.A_0359_KL_3361_1002_1_Ch_Oscilloscope.Channel_1.Data_Out_10 <-> Channel 1/Data Out 10
//   PLC/PLC Instance <-> EtherCAT Master BKCUCX/TcTerminals210_EK1100_1/TcTerminals210_1BK1250/A_0360(KL 3361-1004, 1 Ch. Oscilloscope)
//     PlcTask Inputs/GVL_iXlinker.EtherCAT_Master_BKCUCX.TcTerminals210_EK1100_1.TcTerminals210_1BK1250.A_0360_KL_3361_1004_1_Ch_Oscilloscope.Channel_1.State <-> Channel 1/State
//     PlcTask Inputs/GVL_iXlinker.EtherCAT_Master_BKCUCX.TcTerminals210_EK1100_1.TcTerminals210_1BK1250.A_0360_KL_3361_1004_1_Ch_Oscilloscope.Channel_1.Data_In_0 <-> Channel 1/Data In 0
//     PlcTask Inputs/GVL_iXlinker.EtherCAT_Master_BKCUCX.TcTerminals210_EK1100_1.TcTerminals210_1BK1250.A_0360_KL_3361_1004_1_Ch_Oscilloscope.Channel_1.Data_In_1 <-> Channel 1/Data In 1
//     PlcTask Inputs/GVL_iXlinker.EtherCAT_Master_BKCUCX.TcTerminals210_EK1100_1.TcTerminals210_1BK1250.A_0360_KL_3361_1004_1_Ch_Oscilloscope.Channel_1.Data_In_2 <-> Channel 1/Data In 2
//     PlcTask Inputs/GVL_iXlinker.EtherCAT_Master_BKCUCX.TcTerminals210_EK1100_1.TcTerminals210_1BK1250.A_0360_KL_3361_1004_1_Ch_Oscilloscope.Channel_1.Data_In_3 <-> Channel 1/Data In 3
//     PlcTask Inputs/GVL_iXlinker.EtherCAT_Master_BKCUCX.TcTerminals210_EK1100_1.TcTerminals210_1BK1250.A_0360_KL_3361_1004_1_Ch_Oscilloscope.Channel_1.Data_In_4 <-> Channel 1/Data In 4
//     PlcTask Inputs/GVL_iXlinker.EtherCAT_Master_BKCUCX.TcTerminals210_EK1100_1.TcTerminals210_1BK1250.A_0360_KL_3361_1004_1_Ch_Oscilloscope.Channel_1.Data_In_5 <-> Channel 1/Data In 5
//     PlcTask Inputs/GVL_iXlinker.EtherCAT_Master_BKCUCX.TcTerminals210_EK1100_1.TcTerminals210_1BK1250.A_0360_KL_3361_1004_1_Ch_Oscilloscope.Channel_1.Data_In_6 <-> Channel 1/Data In 6
//     PlcTask Inputs/GVL_iXlinker.EtherCAT_Master_BKCUCX.TcTerminals210_EK1100_1.TcTerminals210_1BK1250.A_0360_KL_3361_1004_1_Ch_Oscilloscope.Channel_1.Data_In_7 <-> Channel 1/Data In 7
//     PlcTask Inputs/GVL_iXlinker.EtherCAT_Master_BKCUCX.TcTerminals210_EK1100_1.TcTerminals210_1BK1250.A_0360_KL_3361_1004_1_Ch_Oscilloscope.Channel_1.Data_In_8 <-> Channel 1/Data In 8
//     PlcTask Inputs/GVL_iXlinker.EtherCAT_Master_BKCUCX.TcTerminals210_EK1100_1.TcTerminals210_1BK1250.A_0360_KL_3361_1004_1_Ch_Oscilloscope.Channel_1.Data_In_9 <-> Channel 1/Data In 9
//     PlcTask Inputs/GVL_iXlinker.EtherCAT_Master_BKCUCX.TcTerminals210_EK1100_1.TcTerminals210_1BK1250.A_0360_KL_3361_1004_1_Ch_Oscilloscope.Channel_1.Data_In_10 <-> Channel 1/Data In 10
//     PlcTask Outputs/GVL_iXlinker.EtherCAT_Master_BKCUCX.TcTerminals210_EK1100_1.TcTerminals210_1BK1250.A_0360_KL_3361_1004_1_Ch_Oscilloscope.Channel_1.Ctrl <-> Channel 1/Ctrl
//     PlcTask Outputs/GVL_iXlinker.EtherCAT_Master_BKCUCX.TcTerminals210_EK1100_1.TcTerminals210_1BK1250.A_0360_KL_3361_1004_1_Ch_Oscilloscope.Channel_1.Data_Out_0 <-> Channel 1/Data Out 0
//     PlcTask Outputs/GVL_iXlinker.EtherCAT_Master_BKCUCX.TcTerminals210_EK1100_1.TcTerminals210_1BK1250.A_0360_KL_3361_1004_1_Ch_Oscilloscope.Channel_1.Data_Out_1 <-> Channel 1/Data Out 1
//     PlcTask Outputs/GVL_iXlinker.EtherCAT_Master_BKCUCX.TcTerminals210_EK1100_1.TcTerminals210_1BK1250.A_0360_KL_3361_1004_1_Ch_Oscilloscope.Channel_1.Data_Out_2 <-> Channel 1/Data Out 2
//     PlcTask Outputs/GVL_iXlinker.EtherCAT_Master_BKCUCX.TcTerminals210_EK1100_1.TcTerminals210_1BK1250.A_0360_KL_3361_1004_1_Ch_Oscilloscope.Channel_1.Data_Out_3 <-> Channel 1/Data Out 3
//     PlcTask Outputs/GVL_iXlinker.EtherCAT_Master_BKCUCX.TcTerminals210_EK1100_1.TcTerminals210_1BK1250.A_0360_KL_3361_1004_1_Ch_Oscilloscope.Channel_1.Data_Out_4 <-> Channel 1/Data Out 4
//     PlcTask Outputs/GVL_iXlinker.EtherCAT_Master_BKCUCX.TcTerminals210_EK1100_1.TcTerminals210_1BK1250.A_0360_KL_3361_1004_1_Ch_Oscilloscope.Channel_1.Data_Out_5 <-> Channel 1/Data Out 5
//     PlcTask Outputs/GVL_iXlinker.EtherCAT_Master_BKCUCX.TcTerminals210_EK1100_1.TcTerminals210_1BK1250.A_0360_KL_3361_1004_1_Ch_Oscilloscope.Channel_1.Data_Out_6 <-> Channel 1/Data Out 6
//     PlcTask Outputs/GVL_iXlinker.EtherCAT_Master_BKCUCX.TcTerminals210_EK1100_1.TcTerminals210_1BK1250.A_0360_KL_3361_1004_1_Ch_Oscilloscope.Channel_1.Data_Out_7 <-> Channel 1/Data Out 7
//     PlcTask Outputs/GVL_iXlinker.EtherCAT_Master_BKCUCX.TcTerminals210_EK1100_1.TcTerminals210_1BK1250.A_0360_KL_3361_1004_1_Ch_Oscilloscope.Channel_1.Data_Out_8 <-> Channel 1/Data Out 8
//     PlcTask Outputs/GVL_iXlinker.EtherCAT_Master_BKCUCX.TcTerminals210_EK1100_1.TcTerminals210_1BK1250.A_0360_KL_3361_1004_1_Ch_Oscilloscope.Channel_1.Data_Out_9 <-> Channel 1/Data Out 9
//     PlcTask Outputs/GVL_iXlinker.EtherCAT_Master_BKCUCX.TcTerminals210_EK1100_1.TcTerminals210_1BK1250.A_0360_KL_3361_1004_1_Ch_Oscilloscope.Channel_1.Data_Out_10 <-> Channel 1/Data Out 10
//   PLC/PLC Instance <-> EtherCAT Master BKCUCX/TcTerminals210_EK1100_1/TcTerminals210_1BK1250/A_0361(KL 3361-1005, 1 Ch. Oscilloscope)
//     PlcTask Inputs/GVL_iXlinker.EtherCAT_Master_BKCUCX.TcTerminals210_EK1100_1.TcTerminals210_1BK1250.A_0361_KL_3361_1005_1_Ch_Oscilloscope.Channel_1.State <-> Channel 1/State
//     PlcTask Inputs/GVL_iXlinker.EtherCAT_Master_BKCUCX.TcTerminals210_EK1100_1.TcTerminals210_1BK1250.A_0361_KL_3361_1005_1_Ch_Oscilloscope.Channel_1.Data_In_0 <-> Channel 1/Data In 0
//     PlcTask Inputs/GVL_iXlinker.EtherCAT_Master_BKCUCX.TcTerminals210_EK1100_1.TcTerminals210_1BK1250.A_0361_KL_3361_1005_1_Ch_Oscilloscope.Channel_1.Data_In_1 <-> Channel 1/Data In 1
//     PlcTask Inputs/GVL_iXlinker.EtherCAT_Master_BKCUCX.TcTerminals210_EK1100_1.TcTerminals210_1BK1250.A_0361_KL_3361_1005_1_Ch_Oscilloscope.Channel_1.Data_In_2 <-> Channel 1/Data In 2
//     PlcTask Inputs/GVL_iXlinker.EtherCAT_Master_BKCUCX.TcTerminals210_EK1100_1.TcTerminals210_1BK1250.A_0361_KL_3361_1005_1_Ch_Oscilloscope.Channel_1.Data_In_3 <-> Channel 1/Data In 3
//     PlcTask Inputs/GVL_iXlinker.EtherCAT_Master_BKCUCX.TcTerminals210_EK1100_1.TcTerminals210_1BK1250.A_0361_KL_3361_1005_1_Ch_Oscilloscope.Channel_1.Data_In_4 <-> Channel 1/Data In 4
//     PlcTask Inputs/GVL_iXlinker.EtherCAT_Master_BKCUCX.TcTerminals210_EK1100_1.TcTerminals210_1BK1250.A_0361_KL_3361_1005_1_Ch_Oscilloscope.Channel_1.Data_In_5 <-> Channel 1/Data In 5
//     PlcTask Inputs/GVL_iXlinker.EtherCAT_Master_BKCUCX.TcTerminals210_EK1100_1.TcTerminals210_1BK1250.A_0361_KL_3361_1005_1_Ch_Oscilloscope.Channel_1.Data_In_6 <-> Channel 1/Data In 6
//     PlcTask Inputs/GVL_iXlinker.EtherCAT_Master_BKCUCX.TcTerminals210_EK1100_1.TcTerminals210_1BK1250.A_0361_KL_3361_1005_1_Ch_Oscilloscope.Channel_1.Data_In_7 <-> Channel 1/Data In 7
//     PlcTask Inputs/GVL_iXlinker.EtherCAT_Master_BKCUCX.TcTerminals210_EK1100_1.TcTerminals210_1BK1250.A_0361_KL_3361_1005_1_Ch_Oscilloscope.Channel_1.Data_In_8 <-> Channel 1/Data In 8
//     PlcTask Inputs/GVL_iXlinker.EtherCAT_Master_BKCUCX.TcTerminals210_EK1100_1.TcTerminals210_1BK1250.A_0361_KL_3361_1005_1_Ch_Oscilloscope.Channel_1.Data_In_9 <-> Channel 1/Data In 9
//     PlcTask Inputs/GVL_iXlinker.EtherCAT_Master_BKCUCX.TcTerminals210_EK1100_1.TcTerminals210_1BK1250.A_0361_KL_3361_1005_1_Ch_Oscilloscope.Channel_1.Data_In_10 <-> Channel 1/Data In 10
//     PlcTask Outputs/GVL_iXlinker.EtherCAT_Master_BKCUCX.TcTerminals210_EK1100_1.TcTerminals210_1BK1250.A_0361_KL_3361_1005_1_Ch_Oscilloscope.Channel_1.Ctrl <-> Channel 1/Ctrl
//     PlcTask Outputs/GVL_iXlinker.EtherCAT_Master_BKCUCX.TcTerminals210_EK1100_1.TcTerminals210_1BK1250.A_0361_KL_3361_1005_1_Ch_Oscilloscope.Channel_1.Data_Out_0 <-> Channel 1/Data Out 0
//     PlcTask Outputs/GVL_iXlinker.EtherCAT_Master_BKCUCX.TcTerminals210_EK1100_1.TcTerminals210_1BK1250.A_0361_KL_3361_1005_1_Ch_Oscilloscope.Channel_1.Data_Out_1 <-> Channel 1/Data Out 1
//     PlcTask Outputs/GVL_iXlinker.EtherCAT_Master_BKCUCX.TcTerminals210_EK1100_1.TcTerminals210_1BK1250.A_0361_KL_3361_1005_1_Ch_Oscilloscope.Channel_1.Data_Out_2 <-> Channel 1/Data Out 2
//     PlcTask Outputs/GVL_iXlinker.EtherCAT_Master_BKCUCX.TcTerminals210_EK1100_1.TcTerminals210_1BK1250.A_0361_KL_3361_1005_1_Ch_Oscilloscope.Channel_1.Data_Out_3 <-> Channel 1/Data Out 3
//     PlcTask Outputs/GVL_iXlinker.EtherCAT_Master_BKCUCX.TcTerminals210_EK1100_1.TcTerminals210_1BK1250.A_0361_KL_3361_1005_1_Ch_Oscilloscope.Channel_1.Data_Out_4 <-> Channel 1/Data Out 4
//     PlcTask Outputs/GVL_iXlinker.EtherCAT_Master_BKCUCX.TcTerminals210_EK1100_1.TcTerminals210_1BK1250.A_0361_KL_3361_1005_1_Ch_Oscilloscope.Channel_1.Data_Out_5 <-> Channel 1/Data Out 5
//     PlcTask Outputs/GVL_iXlinker.EtherCAT_Master_BKCUCX.TcTerminals210_EK1100_1.TcTerminals210_1BK1250.A_0361_KL_3361_1005_1_Ch_Oscilloscope.Channel_1.Data_Out_6 <-> Channel 1/Data Out 6
//     PlcTask Outputs/GVL_iXlinker.EtherCAT_Master_BKCUCX.TcTerminals210_EK1100_1.TcTerminals210_1BK1250.A_0361_KL_3361_1005_1_Ch_Oscilloscope.Channel_1.Data_Out_7 <-> Channel 1/Data Out 7
